// TwinCAT 3 PLC project TEXXX_XXX
// ProgramVersion: 3.1.4024.0
// libraries:
//   Tc2_Standard, * (Beckhoff Automation GmbH)
//   Tc2_System, * (Beckhoff Automation GmbH)
//   Tc2_Utilities, * (Beckhoff Automation GmbH)
//   Tc3_Module, * (Beckhoff Automation GmbH)
// project tree:
//   DUTs/HMI/ ST_StatusBanner.TcDUT (not stored)
//   DUTs/IO/CARDS/ ST_Terminal_Info.TcDUT, ST_EL1809.TcDUT, ST_EL2809.TcDUT
//   DUTs/MASTER/ E_MachineState.TcDUT, E_ProcessCycle.TcDUT, ST_ButtonsLamps.TcDUT (not stored), ST_HMI_IO.TcDUT, ST_MachineStatus.TcDUT, ST_MasterCTRL.TcDUT, ST_StationCMD.TcDUT, ST_StationStatus.TcDUT (not stored), ST_Puls.TcDUT (not stored), ST_StatisticsHMI.TcDUT (not stored)
//   DUTs/MASTER/log_CSV/ ST_CSVProcess.TcDUT, ST_UserLog.TcDUT (not stored), ST_CycleData.TcDUT
//   DUTs/STATIONS/STATION_1/ E_Station1_State.TcDUT, ST_CycleDataStation1.TcDUT, ST_Station_1.TcDUT
//   DUTs/STATIONS/STATION_2/ E_Station2_State.TcDUT, ST_CycleDataStation2.TcDUT, ST_Station_2.TcDUT
//   DUTs/STATIONS/STATION_3/ E_Station3_State.TcDUT, ST_CycleDataStation3.TcDUT, ST_Station_3.TcDUT
//   DUTs/USER_ALARMS_EVENTS/EVENTS/ ST_ActiveEvents.TcDUT (not stored), ST_EventsAssigment.TcDUT, ST_EventsAssigmentGeneral.TcDUT, ST_EventsHistory.TcDUT, ST_EVENT.TcDUT, ST_StationEvents.TcDUT
//   DUTs/USER_ALARMS_EVENTS/ ST_UserLogHMI.TcDUT (not stored)
//   GVLs/ GVL_Constants.TcGVL, GVL_HMI.TcGVL, GVL_IO.TcGVL, GVL_Master.TcGVL, GVL_Persistent.TcGVL, GVL_Stations.TcGVL
//   / PlcTask.TcTTO (not stored)
//   POUs/A_MASTER/ A_1_PRG_Main_Master.TcPOU, A_2_PRG_MachineCtrl.TcPOU, A_3_PRG_FaultHandling.TcPOU, A_4_PRG_MasterSystemTime.TcPOU
//   POUs/B_STATIONS/B_1_STATION_1/ B_1_1_PRG_Master_Station_1.TcPOU
//   POUs/B_STATIONS/B_2_STATION_2/ B_2_1_PRG_Master_Station_2.TcPOU
//   POUs/B_STATIONS/B_3_STATION_3/ B_3_1_PRG_Master_Station_3.TcPOU
//   POUs/C_HMI/ C_1_PRG_MainHMI.TcPOU
//   POUs/D_CSV/ D_1_WriteDataToCSV.TcPOU
//   POUs/ MAIN.TcPOU
//   POUs/Utilities/ FB_EventsManager.TcPOU, FB_UserLog.TcPOU, FB_Pulse.TcPOU (not stored), FB_TerminalInfo.TcPOU, FB_TimeControl.TcPOU, PRG_Puls.TcPOU (not stored)
// real-time tasks:
//   TASK PlcTask: cycle T#10ms, priority 20, ADS port 350

// ---- DUTs/IO/CARDS/ST_Terminal_Info.TcDUT
TYPE ST_Terminal_Info :
STRUCT
	
	nTerminal_State                        AT %I*			:    UINT;	// Terminal State from IO Terminal Info Data
	sTerminalInfo                                           :    STRING;
    fbTerminalInfo                                          :    FB_TerminalInfo;
END_STRUCT
END_TYPE

// ---- DUTs/IO/CARDS/ST_EL1809.TcDUT
TYPE ST_EL1809 :
STRUCT
	//--------------------------------------------------------------------------------------------------------
	sTerminalName                                           :   STRING(200):= 'EL1809 | 16-Channel Digital Input';
    //============================================================================================================================	
	// TERMINAL - EL1809 16-Channel Digital Input Terminal 	
	iEL1809_Ch1                				AT %I*			: 	BOOL;	// EL1809 channel 1
	iEL1809_Ch2                   			AT %I*			: 	BOOL;	// EL1809 channel 2
	iEL1809_Ch3        						AT %I*	 		: 	BOOL;	// EL1809 channel 3
	iEL1809_Ch4   							AT %I*	 		: 	BOOL;	// EL1809 channel 4
	iEL1809_Ch5         				 	AT %I*	 		: 	BOOL;	// EL1809 channel 5 		     			
	iEL1809_Ch6 							AT %I*			: 	BOOL;	// EL1809 channel 6
	iEL1809_Ch7               				AT %I*          :   BOOL;   // EL1809 channel 7 
    iEL1809_Ch8          					AT %I*          :   BOOL;   // EL1809 channel 8
    iEL1809_Ch9           					AT %I*          :   BOOL;   // EL1809 channel 9
	iEL1809_Ch10                			AT %I*          :   BOOL;   // EL1809 channel 10
	iEL1809_Ch11                    		AT %I*          :   BOOL;   // EL1809 channel 11
	iEL1809_Ch12                          	AT %I*          :   BOOL;   // EL1809 channel 12	   
	iEL1809_Ch13         		    		AT %I*	 		: 	BOOL;	// EL1809 channel 13   
	iEL1809_Ch14       						AT %I*	 		: 	BOOL;	// EL1809 channel 14 
	iEL1809_Ch15							AT %I*			: 	BOOL;	// EL1809 channel 15  
	iEL1809_Ch16							AT %I*	 		: 	BOOL;	// EL1809 channel 16  	
	
	stTerminalInfo											: 	ST_Terminal_Info;

END_STRUCT
END_TYPE

// ---- DUTs/IO/CARDS/ST_EL2809.TcDUT
TYPE ST_EL2809 :
STRUCT
	//--------------------------------------------------------------------------------------------------------
	sTerminalName                                           :   STRING(200):= 'EL2809 | 16-Channel Digital Output';
	//=============================================================================================================
	// TERMINAL - EL2809	16-Channel Digital Output Terminal	 (Term ...)
	qiEL2809_Ch1 							AT %Q*			: 	BOOL;	// EL2809 channel 1
	qiEL2809_Ch2							AT %Q* 			: 	BOOL;	// EL2809 channel 2
	qiEL2809_Ch3             				AT %Q*	 		: 	BOOL;	// EL2809 channel 3 			
	qiEL2809_Ch4      						AT %Q*	 		: 	BOOL;	// EL2809 channel 4 
	qiEL2809_Ch5  							AT %Q*	 		: 	BOOL;	// EL2809 channel 5
	qiEL2809_Ch6 							AT %Q*	 		: 	BOOL;	// EL2809 channel 6 	
	qiEL2809_Ch7         		    		AT %Q*			: 	BOOL;	// EL2809 channel 7	
	qiEL2809_Ch8							AT %Q*	 		: 	BOOL;	// EL2809 channel 8	
	qiEL2809_Ch9                 			AT %Q*          :   BOOL;   // EL2809 channel 9
	qiEL2809_Ch10             				AT %Q*          :   BOOL;   // EL2809 channel 10   	
	qiEL2809_Ch11     						AT %Q*	 		: 	BOOL;	// EL2809 channel 11	
	qiEL2809_Ch12   						AT %Q*	 		: 	BOOL;	// EL2809 channel 12 
    qiEL2809_Ch13 			        		AT %Q*	 		: 	BOOL;	// EL2809 channel 13 
	qiEL2809_Ch14                 			AT %Q*	 		: 	BOOL;	// EL2809 channel 14 
	qiEL2809_Ch15							AT %Q*	 		: 	BOOL;	// EL2809 channel 15 
    qiEL2809_Ch16         		        	AT %Q*	 		: 	BOOL;	// EL2809 channel 16  
	
	stTerminalInfo											: 	ST_Terminal_Info;
	
END_STRUCT
END_TYPE

// ---- DUTs/MASTER/E_MachineState.TcDUT
{attribute 'qualified_only'}
{attribute 'strict'}
TYPE E_MachineState :
(
	SYSTEM_POWER_UP			:=0,
	IMMEDIATE_STOPPED		:=100,
	SYSTEM_INITIALISING		:=110,
	SYSTEM_READY_TO_START	:=120,
	SYSTEM_AUTO_CYCLE		:=130,
	SYSTEM_STANDBY			:=140,
	STOPPING				:=150,
	CYCLE_STOPPED			:=160,
	MANUAL_MODE				:=170,
	IMMEDIATE_FAULT			:=190,
	CYCLE_STOP_FAULT		:=200
);
END_TYPE

// ---- DUTs/MASTER/E_ProcessCycle.TcDUT
{attribute 'qualified_only'}
{attribute 'strict'}
TYPE E_ProcessCycle :
(

	
IDLE								:=0,
STATION1_MOV1						:=10,
WAIT_STATION1_MOV1					:=20,
STATION2_MOV2						:=30,
WAIT_STATION2_MOV2					:=40,
STATION3_MOV3						:=50,
WAIT_STATION3_MOV3					:=60,
STATION1_MOV3_STATION2_MOV2			:=70,
WAIT_STATION1_MOV3_STATION2_MOV2	:=80,
SAVE_DATA							:=90,
SAVE_DATA2							:=100,
CSV									:=110,

RESET_ALL_CMD						:=120

);
END_TYPE

// ---- DUTs/MASTER/log_CSV/ST_CSVProcess.TcDUT
TYPE ST_CSVProcess :
STRUCT
	
	//INPUTS
	bWriteData			: BOOL;
	sFileNamePath		: STRING(255);
	sDate				: STRING(255);
	aDataHistoryArrayLength : DINT;
	nMAX_CSV_ROWS		: UDINT;
	nMAX_CSV_COLUMNS	: UDINT;
	nDataHistoryIndex	: DINT;
	

	//OUTPUTS
	bError				: BOOL;
	bBusy				: BOOL;
	bDataWrited			: BOOL;
	
	
	
	
END_STRUCT
END_TYPE

// ---- DUTs/MASTER/log_CSV/ST_CycleData.TcDUT
TYPE ST_CycleData :
STRUCT
//-----------------------------------------------------------------------------------GENERAL------------------------------------------------------------------------------------//	

	bPass				: BOOL;
	bFail				: BOOL;	
	sData				: STRING;	
	sTime				: STRING;
	
//-----------------------------------------------------------------------------------STATION 1------------------------------------------------------------------------------------//
/////////////////////////////////////////////////////////////////////////////////////SETTINGS/////////////////////////////////////////////////////////////////////////////////////			
(**************************************************************************CURRENT SETTINGS DURING CYCLE. VELOCITY FOR EXAMPLE****************************************************)	
	
	sSetting1_1			: STRING;	
	nSetting2_1			: DINT;
	bSetting3_1			: BOOL;
	
/////////////////////////////////////////////////////////////////////////////////////GENERAL DATA/////////////////////////////////////////////////////////////////////////////////////			
(**************************************************************************RESULT DATA OF THE CYCLE. DISTANCE FOR EXAMPLE************************************************************)	
	
	sDATA1_1			: STRING;
	nDATA2_1			: DINT;
	bDATA3_1			: BOOL;

////////////////////////////////////////////////////////////////////////////////////RESULTS////////////////////////////////////////////////////////////////////////////////////////
(**************************************************************************DETERMINE IF THE PART FAIL OR PASS*********************************************************************)

	bPass_1				: BOOL;
	bFail_1				: BOOL;		


	
	
	
//-----------------------------------------------------------------------------------STATION 2------------------------------------------------------------------------------------//
/////////////////////////////////////////////////////////////////////////////////////SETTINGS/////////////////////////////////////////////////////////////////////////////////////			
(**************************************************************************CURRENT SETTINGS DURING CYCLE. VELOCITY FOR EXAMPLE****************************************************)	
	
	sSetting1_2			: STRING;	
	nSetting2_2			: DINT;
	bSetting3_2			: BOOL;
	
/////////////////////////////////////////////////////////////////////////////////////GENERAL DATA/////////////////////////////////////////////////////////////////////////////////////			
(**************************************************************************RESULT DATA OF THE CYCLE. DISTANCE FOR EXAMPLE************************************************************)	
	
	sDATA1_2			: STRING;
	nDATA2_2			: DINT;
	bDATA3_2			: BOOL;

////////////////////////////////////////////////////////////////////////////////////RESULTS////////////////////////////////////////////////////////////////////////////////////////
(**************************************************************************DETERMINE IF THE PART FAIL OR PASS*********************************************************************)

	bPass_2				: BOOL;
	bFail_2				: BOOL;		
	
	
	
	
	
//-----------------------------------------------------------------------------------STATION 3------------------------------------------------------------------------------------//
/////////////////////////////////////////////////////////////////////////////////////SETTINGS/////////////////////////////////////////////////////////////////////////////////////			
(**************************************************************************CURRENT SETTINGS DURING CYCLE. VELOCITY FOR EXAMPLE****************************************************)	
	
	sSetting1_3			: STRING;	
	nSetting2_3			: DINT;
	bSetting3_3			: BOOL;
	
/////////////////////////////////////////////////////////////////////////////////////GENERAL DATA/////////////////////////////////////////////////////////////////////////////////////			
(**************************************************************************RESULT DATA OF THE CYCLE. DISTANCE FOR EXAMPLE************************************************************)	
	
	sDATA1_3			: STRING;
	nDATA2_3			: DINT;
	bDATA3_3			: BOOL;

////////////////////////////////////////////////////////////////////////////////////RESULTS////////////////////////////////////////////////////////////////////////////////////////
(**************************************************************************DETERMINE IF THE PART FAIL OR PASS*********************************************************************)

	bPass_3				: BOOL;
	bFail_3				: BOOL;		
	



	
	
END_STRUCT
END_TYPE

// ---- DUTs/MASTER/ST_HMI_IO.TcDUT
TYPE ST_HMI_IO :
STRUCT
	
	bTriggerButtonA				:BOOL;
	bTriggerButtonB				:BOOL;
	bTriggerButtonC				:BOOL;
	
	bOutPutSigA					:BOOL;
	bOutPutSigB					:BOOL;
	bOutPutSigC					:BOOL;
	
END_STRUCT
END_TYPE

// ---- DUTs/MASTER/ST_MachineStatus.TcDUT
TYPE ST_MachineStatus :
STRUCT
	////////////////////////////:
	eMachineState				:E_MachineState;
	
	// Status Flags:
	bSystemPowerUp 				:BOOL;
	bImmediateStopped 			:BOOL;
	bInitialising 				:BOOL;
	bReadyToStart 				:BOOL;
	bAutoCycle 					:BOOL;
	bStandby					:BOOL;
	bStopping					:BOOL;	
	bCycleStopped 				:BOOL;
	bImmediateFault 			:BOOL;
	bCycleStopFault 			:BOOL;
	bManualMode					:BOOL;

END_STRUCT
END_TYPE

// ---- DUTs/MASTER/ST_MasterCTRL.TcDUT
TYPE ST_MasterCTRL :
STRUCT
	

	// Request Flags
	bManualModeRequest					:BOOL;
	
	bCycleStopRequest					:BOOL;
	
	bNoImmediateFault					:BOOL;
	bNoCycleStopFault					:BOOL;


	// Feedback Flags
	bAllStationsReady					:BOOL;
	bAllStationsStopped					:BOOL;
	
	bPowerUpTimerComplete				:BOOL;

	
//-------------------------------------------------------------------------------oldschoo1
		
END_STRUCT
END_TYPE

// ---- DUTs/MASTER/ST_StationCMD.TcDUT
TYPE ST_StationCMD :
STRUCT
//Universal Module CMD Struct

    bEnable       			:BOOL;	// Request module to activate devices
	bExecute				:BOOL;	// Request module to execute CMD
    bReset        			:BOOL;	// Request module to reset error or state
    bAbort        			:BOOL;	// Emergency stop or cancel current task
	bReady					:BOOL;	// Get ready
	bEndCycle				:BOOL; // End cycle
	
	nTaskID       			:UINT;	// Request a Task by its ID	
    bManualMode   			:BOOL;	// Request Manual Mode(jog mode)
	
	
END_STRUCT
END_TYPE

// ---- DUTs/STATIONS/STATION_1/E_Station1_State.TcDUT
{attribute 'qualified_only'}
{attribute 'strict'}
TYPE E_Station1_State :
(
	//GENERIC
	ABORTED				:=10,
	RESET_ERROR			:=20,
	HOMING				:=30,
	READY				:=40,
	//MANUAL_MODE		:=50, /manual mode not needed.
	ERROR				:=60,
	PERSISTENT_ERROR	:=70,
	STOPPING			:=80,
	//SPECIFIC FOR EVERY STATION
	MOVEMENT_A			:=100,
	MOVEMENT_B			:=120,
	MOVEMENT_C			:=130,
	DONE				:=140,
	RESULTS				:=160,
	RESET				:=180
);
END_TYPE

// ---- DUTs/STATIONS/STATION_1/ST_CycleDataStation1.TcDUT
TYPE ST_CycleDataStation1 :
STRUCT
	/////////////////////////////////////////////////////////////////////////////////////SETTINGS/////////////////////////////////////////////////////////////////////////////////////			
(**************************************************************************CURRENT SETTINGS DURING CYCLE. VELOCITY FOR EXAMPLE****************************************************)	
	
	sSetting1			: STRING;	
	nSetting2			: DINT;
	bSetting3			: BOOL;
	
/////////////////////////////////////////////////////////////////////////////////////GENERAL DATA/////////////////////////////////////////////////////////////////////////////////////			
(**************************************************************************RESULT DATA OF THE CYCLE. DISTANCE FOR EXAMPLE************************************************************)	
	
	sDATA1				: STRING;
	nDATA2				: DINT;
	bDATA3				: BOOL;

////////////////////////////////////////////////////////////////////////////////////RESULTS////////////////////////////////////////////////////////////////////////////////////////
(**************************************************************************DETERMINE IF THE PART FAIL OR PASS*********************************************************************)

	bPass				: BOOL;
	bFail				: BOOL;		

END_STRUCT
END_TYPE

// ---- DUTs/STATIONS/STATION_1/ST_Station_1.TcDUT
TYPE ST_Station_1 :
STRUCT
	
	Mov1				: BOOL;		
	Mov2				: BOOL;	
	Mov3				: BOOL;		
	
END_STRUCT
END_TYPE

// ---- DUTs/STATIONS/STATION_2/E_Station2_State.TcDUT
{attribute 'qualified_only'}
{attribute 'strict'}
TYPE E_Station2_State :
(
		//GENERIC
	ABORTED				:=10,
	RESET_ERROR			:=20,
	HOMING				:=30,
	READY				:=40,
	//MANUAL_MODE			:=50, /manual mode not needed.
	ERROR				:=60,
	PERSISTENT_ERROR	:=70,
	STOPPING			:=80,
	//SPECIFIC FOR EVERY STATION
	MOVEMENT_A			:=100,
	MOVEMENT_B			:=120,
	MOVEMENT_C			:=130,
	DONE				:=140,
	RESULTS				:=160,
	RESET				:=180
);
END_TYPE

// ---- DUTs/STATIONS/STATION_2/ST_CycleDataStation2.TcDUT
TYPE ST_CycleDataStation2 :
STRUCT
	/////////////////////////////////////////////////////////////////////////////////////SETTINGS/////////////////////////////////////////////////////////////////////////////////////			
(**************************************************************************CURRENT SETTINGS DURING CYCLE. VELOCITY FOR EXAMPLE****************************************************)	
	
	sSetting1			: STRING;	
	nSetting2			: DINT;
	bSetting3			: BOOL;
	
/////////////////////////////////////////////////////////////////////////////////////GENERAL DATA/////////////////////////////////////////////////////////////////////////////////////			
(**************************************************************************RESULT DATA OF THE CYCLE. DISTANCE FOR EXAMPLE************************************************************)	
	
	sDATA1				: STRING;
	nDATA2				: DINT;
	bDATA3				: BOOL;

////////////////////////////////////////////////////////////////////////////////////RESULTS////////////////////////////////////////////////////////////////////////////////////////
(**************************************************************************DETERMINE IF THE PART FAIL OR PASS*********************************************************************)

	bPass				: BOOL;
	bFail				: BOOL;		

END_STRUCT
END_TYPE

// ---- DUTs/STATIONS/STATION_2/ST_Station_2.TcDUT
TYPE ST_Station_2 :
STRUCT
	
	Mov1				: BOOL;		
	Mov2				: BOOL;	
	Mov3				: BOOL;		
	
END_STRUCT
END_TYPE

// ---- DUTs/STATIONS/STATION_3/E_Station3_State.TcDUT
{attribute 'qualified_only'}
{attribute 'strict'}
TYPE E_Station3_State :
(
		//GENERIC
	ABORTED				:=10,
	RESET_ERROR			:=20,
	HOMING				:=30,
	READY				:=40,
	//MANUAL_MODE			:=50, /manual mode not needed.
	ERROR				:=60,
	PERSISTENT_ERROR	:=70,
	STOPPING			:=80,
	//SPECIFIC FOR EVERY STATION
	MOVEMENT_A			:=100,
	MOVEMENT_B			:=120,
	MOVEMENT_C			:=130,
	DONE				:=140,
	RESULTS				:=160,
	RESET				:=180
);
END_TYPE

// ---- DUTs/STATIONS/STATION_3/ST_CycleDataStation3.TcDUT
TYPE ST_CycleDataStation3 :
STRUCT
	/////////////////////////////////////////////////////////////////////////////////////SETTINGS/////////////////////////////////////////////////////////////////////////////////////			
(**************************************************************************CURRENT SETTINGS DURING CYCLE. VELOCITY FOR EXAMPLE****************************************************)	
	
	sSetting1			: STRING;	
	nSetting2			: DINT;
	bSetting3			: BOOL;
	
/////////////////////////////////////////////////////////////////////////////////////GENERAL DATA/////////////////////////////////////////////////////////////////////////////////////			
(**************************************************************************RESULT DATA OF THE CYCLE. DISTANCE FOR EXAMPLE************************************************************)	
	
	sDATA1				: STRING;
	nDATA2				: DINT;
	bDATA3				: BOOL;

////////////////////////////////////////////////////////////////////////////////////RESULTS////////////////////////////////////////////////////////////////////////////////////////
(**************************************************************************DETERMINE IF THE PART FAIL OR PASS*********************************************************************)

	bPass				: BOOL;
	bFail				: BOOL;		

END_STRUCT
END_TYPE

// ---- DUTs/STATIONS/STATION_3/ST_Station_3.TcDUT
TYPE ST_Station_3 :
STRUCT
	
	Mov1				: BOOL;		
	Mov2				: BOOL;	
	Mov3				: BOOL;		
	
END_STRUCT
END_TYPE

// ---- DUTs/USER_ALARMS_EVENTS/EVENTS/ST_EventsAssigment.TcDUT
TYPE ST_EventsAssigment :
STRUCT
	
	sEventText							: STRING(255);
	sSolution							: STRING(255);
END_STRUCT
END_TYPE

// ---- DUTs/USER_ALARMS_EVENTS/EVENTS/ST_EventsAssigmentGeneral.TcDUT
TYPE ST_EventsAssigmentGeneral :
STRUCT
	
	astImmediateFaultEvents				: ARRAY [1..100] OF ST_EventsAssigment;
	astCycleStopFaultEvents				: ARRAY [1..100] OF ST_EventsAssigment;
	astCycleStopRequestEvents			: ARRAY [1..100] OF ST_EventsAssigment;
	astMessage							: ARRAY [1..100] OF ST_EventsAssigment;
	
	
END_STRUCT
END_TYPE

// ---- DUTs/USER_ALARMS_EVENTS/EVENTS/ST_EventsHistory.TcDUT
TYPE ST_EventsHistory :
STRUCT
	
	sEventTex									: STRING(255);
	sType										: STRING(255);
	sDate										: STRING(255);
	sTime										: STRING(255);
	abType										: DINT;					//1:Alarm
																		//2:Alert
																		//3:Message
	
END_STRUCT
END_TYPE

// ---- DUTs/USER_ALARMS_EVENTS/EVENTS/ST_EVENT.TcDUT
TYPE ST_EVENT :
STRUCT
	
	bImmediateFault						: BOOL;
	bCycleStopFault						: BOOL;
	bCycleStopRequest					: BOOL;
	bMessage							: BOOL;
	
	bAssignedID							: DINT;
	
	bEventFlag							: BOOL;
	bEventTimer							: TON;
	bEventText							: STRING(255);
	bEventTextHMI						: STRING(255);
	sSolution							: STRING(255);
	bActive								: BOOL;

END_STRUCT
END_TYPE

// ---- DUTs/USER_ALARMS_EVENTS/EVENTS/ST_StationEvents.TcDUT
TYPE ST_StationEvents :
STRUCT
	
	aEvents								: ARRAY [0..100] OF ST_EVENT;	
	
	bImmediateFault						: BOOL;
	bCycleStopFault						: BOOL;
	bCycleStopRequest					: BOOL;
			
END_STRUCT
END_TYPE

// ---- GVLs/GVL_Constants.TcGVL
VAR_GLOBAL CONSTANT
////////////////////////////////////////:	///////////////////////////////////////////////////
/////////////////////////////////////////////////////////////////////////////////////HMI/////////////////////////////////////////////////////////////////////////////////////
	
    sWHITE                              :   STRING(40)  := '{"color":"rgba(255,255,255,255)"}';
    sBLACK                              :   STRING(40)  := '{"color":"rgba(0,0,0,1)"}';
    sYELLOW                             :   STRING(40)  := '{"color":"rgba(255,255,0,1)"}';
    sGREEN                             	:   STRING(40)  := '{"color":"rgba(70,166,63,1)"}';
	sLGREEN                             :   STRING(40)  := '{"color":"rgba(58,211,20,1)"}';
    sORANGE                             :   STRING(40)  := '{"color":"rgba(255,153,51,1)"}';
    sNYPROORANGE                        :   STRING(40)  := '{"color":"rgba(255,140,0,1)"}';
    sRED                                :   STRING(40)  := '{"color":"rgba(255,0,0,1)"}';
	sLRED                               :   STRING(40)  := '{"color":"rgba(233,53,44,1)"}';
    sBLUE                               :   STRING(40)  := '{"color":"rgba(0,0,255,1)"}';
	sLBLUE                              :   STRING(40)  := '{"color":"rgba(0,162,232,1)"}';
    sGREY                               :   STRING(40)  := '{"color":"rgba(164,158,158,1)"}';
    sScreenGREY                         :   STRING(40)  := '{"color":"rgba(225,225,225,1)"}';
    sDARKGREY                           :   STRING(40)  := '{"color":"rgba(50,50,50,1)"}';
    sPURPLE                             :   STRING(40)  := '{"color":"rgba(128,0,128,1)"}';
    sVIOLET                             :   STRING(40)  := '{"color":"rgba(204,153,255,1)"}';
    sTRANSP                             :   STRING(40)  := '{"color":"rgba(255,255,255,0)"}';
    sGREENPass                          :   STRING(40)  := '{"color":"rgba(0,153,51,1)"}';
    sREDFail                            :   STRING(40)  := '{"color":"rgba(244,68,68,255)"}';
    sBLUEInProgress                     :   STRING(40)  := '{"color":"rgba(54,100,221,1)"}';
	sGREENISHTEAColor					:	STRING(40)  := '{"color":"rgba(60,192,134,255)"}'	;		

	nBLACK								: 	DWORD 	:= 	16#FF000000;	 // format: TTRRGGBB where T -> 00 = full transparency and FF = full opaque
	nWHITE								: 	DWORD 	:= 	16#FFFFFFFF;
	nYELLOW								: 	DWORD 	:= 	16#FFFFFF00; 
	nGREEN								: 	DWORD 	:= 	16#FF008A00;
	nLIGHTGREEN                         :   DWORD   :=  16#FF98FB89;
	nORANGE								: 	DWORD 	:= 	16#FFFFA500;
	nNYPROORANGE						:	DWORD	:=	16#FFF05322;
	nRED								: 	DWORD 	:= 	16#FFFF0000;
	nBLUE								: 	DWORD 	:= 	16#FF0000FF;
	nLIGHTBLUE                          :   DWORD   :=  16#FF08ADF4;
	nGREY								: 	DWORD 	:= 	16#FFA9A9A9;	
	nDARKGREY							:	DWORD	:=	16#FF808080;
	nPURPLE								:	DWORD	:=	16#FF800080;
	nVIOLET								:	DWORD	:=	16#FFEE82EE;
	nTRANSP								:	DWORD	:=	16#00FFFFFF;	// full transparent WHITE
	
/////////////////////////////////////////////////////////////////////////////////////CSV/////////////////////////////////////////////////////////////////////////////////////
	
	MAX_CSV_ROWS 						: UDINT := 200;
	MAX_CSV_COLUMNS 					: UDINT := 27;
	MAX_CSV_FIELD_LENGTH				: UDINT := 100;
	
	
	
END_VAR

// ---- GVLs/GVL_HMI.TcGVL
VAR_GLOBAL
////////////////////////////////////////:	///////////////////////////////////////////////////
/////////////////////////////////////////////////////////////////////////////////////GENERIC/////////////////////////////////////////////////////////////////////////////////////

	stHMI_IO							: ST_HMI_IO;
	bQuitHMI							: BOOL;
	bShutDown							: BOOL;
	stStatusBanner						: ST_StatusBanner;
	

/////////////////////////////////////////////////////////////////////////////////////SYSTEM INFO/////////////////////////////////////////////////////////////////////////////////////

	sSoftwareVersion					: STRING := ' 1.0 ';
	sSoftwareDate						: STRING := ' 10.December.2024 ';
	sTC3Version							: STRING := ' v3.1.4024.53, Runtime v3.1.4024.40 ';
	sHMIVersion							: STRING := ' TcXaeShell Version 15.0.28010.2050 D15.8 ';
	sSystemName							: STRING := ' Print & Applay Labeller ' ;
	sProjectID							: STRING := ' TE 1099 PAL' ;
	sAplication                     	: STRING := ' Print & Applay Labeller ';
	sHMIServer                			: STRING := ' ---- ';
	
	NetAmsId        	       			: T_AmsNetId := ''; // AMS-ID for com port setup 
	
/////////////////////////////////////////////////////////////////////////////////////USER LOG/////////////////////////////////////////////////////////////////////////////////////

	sUserGroupIn						: STRING;
	sUserGroupOut						: STRING;
	sUserName							: STRING;
	bUserLoggedIn						: BOOL;			
	bLogOut								: BOOL;	
	rUserLoggedIn						: R_TRIG;

/////////////////////////////////////////////////////////////////////////////////////MANUAL/////////////////////////////////////////////////////////////////////////////////////

	bEnableManual						: BOOL;
	nMainRegion							: DINT;
	bManualModeOffFlag					: BOOL;
	
END_VAR

// ---- GVLs/GVL_IO.TcGVL
VAR_GLOBAL
	
	

	//	dw_T01_EK1100                                                	| EtherCAT Coupler 
	//	dw_T02_EL6070-0033                                           	| EtherCAT Terminal, license key for TwinCAT 3.1
	
	dw_T03_EL1809                                                		: st_EL1809; //16 Channel Digital Input ( 24VDC ) 
	dw_T04_EL2809                                                		: st_EL2809; // 16 Channel Digital Output ( 24VDC )

END_VAR

// ---- GVLs/GVL_Master.TcGVL
VAR_GLOBAL
////////////////////////////////////////:	///////////////////////////////////////////////////
/////////////////////////////////////////////////////////////////////////////////////GENERIC/////////////////////////////////////////////////////////////////////////////////////

	// PowerUP 
	tonSystemPowerUP				:TON;
	tSystemPowerUP_Time				:TIME								:=T#35S;
	bSystemPoweringUP				:BOOL								:=TRUE; //Global System PowerUP Flag
	
	fbSystemShutDown     	        : NT_Shutdown;
	stButtonsLamps					: ST_ButtonsLamps;
	stPuls							: ST_Puls;		

	stCSVProcess					: ST_CSVProcess;
/////////////////////////////////////////////////////////////////////////////////////Event Log/////////////////////////////////////////////////////////////////////////////////////
	
	stStationEvents				: ARRAY[0..3] OF  ST_StationEvents;//0: GENERAL
																	//1: STATION 1
																	//1: STATION 2
																	//3: STATION 3
	astActiveEvents				: ARRAY [0..50] OF ST_ActiveEvents;
	astEventsHistory			: ARRAY[0..200] OF ST_EventsHistory;
	
/////////////////////////////////////////////////////////////////////////////////////MACHINE CONTROL////////////////////////////////////////////////////////////////////////////
	
	stMachineStatus					: ST_MachineStatus;	
	stMasterCtrl					: ST_MasterCTRL;
	bStatisticsTest					: ARRAY[0..6] OF  BOOL;
	
////////////////////////////////////////////////////////////////////////////////////SYSTEM////////////////////////////////////////////////////////////////////////////
	stSystemTime				: TIMESTRUCT;
	sSystemTime					: STRING(255);
	sSystemDate					: STRING(255);
	
	bResetTest								: BOOL;
	tonResetTest							: TON;
	
	stEventsAssigment						: ST_EventsAssigmentGeneral;	
END_VAR

// ---- GVLs/GVL_Persistent.TcGVL

VAR_GLOBAL PERSISTENT
	
/////////////////////////////////////////////////////////////////////////////////////Log/////////////////////////////////////////////////////////////////////////////////////
	
	stUserLog					: ARRAY [0..250] OF ST_UserLog;
	
	stStatisticsHMI				: ARRAY [0..3] OF ST_StatisticsHMI;	//0: GENERAL
																	//1: STATION 1
																	//2: STATION 2
																	//3: STATION 3
	aDataHistory				: ARRAY[0..200] OF ST_CycleData;
	nIndexDataHistory			: DINT;


END_VAR

// ---- GVLs/GVL_Stations.TcGVL
VAR_GLOBAL
/////////////////////////////////////////////////////////////////////////////////////Station 1/////////////////////////////////////////////////////////////////////////////////////
	
	stStation1							: ST_Station_1;
	CMD_Station1						: ST_StationCMD;
	stCycleDataStation1					: ST_CycleDataStation1;
	
/////////////////////////////////////////////////////////////////////////////////////Station 2/////////////////////////////////////////////////////////////////////////////////////

	stStation2							: ST_Station_2;
	CMD_Station2						: ST_StationCMD;
	stCycleDataStation2					: ST_CycleDataStation2;

/////////////////////////////////////////////////////////////////////////////////////Station 3/////////////////////////////////////////////////////////////////////////////////////

	stStation3							: ST_Station_3;	
	CMD_Station3						: ST_StationCMD;
	stCycleDataStation3					: ST_CycleDataStation3;

END_VAR

// ---- POUs/A_MASTER/A_1_PRG_Main_Master.TcPOU
PROGRAM A_1_PRG_Main_Master
VAR
	
	rtrigButton             				: ARRAY[1..3] OF Tc2_Standard.R_TRIG;
	ftrigButton             				: ARRAY[1..3] OF Tc2_Standard.F_TRIG; 
	
	fbStringFormatter       				: Tc2_Utilities.FB_FormatString;
	fbEventsManager							: FB_EventsManager;
	
	ntShutdown								: TC2_Utilities.NT_Shutdown;
	closeChrome 							: NT_StartProcess;
	tonUserLogOut							: TON;
	fbUserLog								: FB_UserLog;
	
	nFindAdm								: INT;
	nFindEng								: INT;
	nFindOpe								: INT;
	sUserGroupName							: STRING (255);
	sAdmGroup								: STRING (255)							:= 'Administrator';
	sEngGroup								: STRING (255)							:= 'Engineer';
	sOpeGroup								: STRING (255)							:= 'Operator';
	
	rEfficency								: STRING(510);
	
	fbSystemTime							: NT_GetTime;
	

	
END_VAR

/////////////////////////////////////////////////////////////////////////////////////GENERAL/////////////////////////////////////////////////////////////////////////////////////
A_3_PRG_FaultHandling();
a_ACT_ButtonsLamps();
d_ACT_ShutdownAndQuit();
e_ACT_UserLog();
f_ACT_TerminalInfo();
g_ACT_Manual();
h_ACT_Statistics();

C_1_PRG_MainHMI();
D_1_WriteDataToCSV();

PRG_Puls();

// System PowerUP CTRL
tonSystemPowerUP(IN:=bSystemPoweringUP, PT:=tSystemPowerUP_Time);
IF tonSystemPowerUP.Q THEN 
bSystemPoweringUP:=FALSE;
END_IF


A_4_PRG_MasterSystemTime();
/////////////////////////////////////////////////////////////////////////////////////STATIONS/////////////////////////////////////////////////////////////////////////////////////

B_1_1_PRG_Master_Station_1(CMD := CMD_Station1);
B_2_1_PRG_Master_Station_2(CMD := CMD_Station2);
B_3_1_PRG_Master_Station_3(CMD := CMD_Station3);

/////////////////////////////////////////////////////////////////////////////////////PROCESS/////////////////////////////////////////////////////////////////////////////////////

A_2_PRG_MachineCtrl();

/////////////////////////////////////////////////////////////////////////////////////EVENT LOG/////////////////////////////////////////////////////////////////////////////////////

fbEventsManager	(			//INPUTS
							bPulse 							:= stPuls.bFlash10Hz, 
							bResetFaults 					:= bResetTest, 
							stStationEvents 				:= stStationEvents,
							sSystemTime						:= sSystemTime,
							sSystemDate						:= sSystemDate,
 							stEventsAssigment				:= stEventsAssigment,
							
							//OUTPUTS
							astActiveEvents 				=> astActiveEvents,
							astEventsHistory				=> astEventsHistory
							);



////////////////////////////////////////////////////////////////////////////////////SYSTEM DATE & TIME/////////////////////////////////////////////////////////////////////////////////////

fbSystemTime( START := stPuls.bFlash10Hz, TIMESTR => stSystemTime);
	

sSystemTime					:= 	CONCAT( STR1 := WORD_TO_STRING(stSystemTime.wHour), STR2 := CONCAT( STR1 := ':', STR2 := 
								CONCAT( STR1 := WORD_TO_STRING(stSystemTime.wMinute), STR2 := 
								CONCAT(STR1 := ':', STR2 := WORD_TO_STRING(stSystemTime.wSecond)))));
								
sSystemDate					:= 	CONCAT( STR1 := WORD_TO_STRING(stSystemTime.wDay), STR2 := 
								CONCAT(STR1 := '/', STR2 := CONCAT(STR1 := WORD_TO_STRING(stSystemTime.wMonth), STR2 := 
								CONCAT(STR1 := '/', STR2 := WORD_TO_STRING(stSystemTime.wYear)))));

ACTION a_ACT_ButtonsLamps:
//===================================================================
stButtonsLamps.bStartButtonFallingEdge 	:= ftrigButton[1].Q ;
stButtonsLamps.bStartButtonRisingEdge 	:= rtrigButton[1].Q ;
stButtonsLamps.bStopButtonFallingEdge 	:= ftrigButton[2].Q ; 
stButtonsLamps.bStopButtonRisingEdge 	:= rtrigButton[2].Q ;  
stButtonsLamps.bResetButtonFallingEdge 	:= ftrigButton[3].Q ;
stButtonsLamps.bResetButtonRisingEdge 	:= rtrigButton[3].Q ;



ftrigButton[1](CLK :=);
rtrigButton[1](CLK						:=);
ftrigButton[2](CLK						:=);
rtrigButton[2](CLK						:=);
ftrigButton[3](CLK	:=bResetTest 		);
rtrigButton[3](CLK						:=);



//GVL_IO.dw_T11_EL2809.qRESETButton_Indicator := stPuls.bFlash2Hz AND (NOT stMachineStatus.bInitialising AND NOT stMachineStatus.bAutoCycle AND NOT stMachineStatus.bManualMode AND NOT stMachineStatus.bReadyToStart) ;
//GVL_IO.dw_T11_EL2809.qStartButton_Indicator := (stPuls.bFlash2Hz AND stMachineStatus.bReadyToStart) OR (stMachineStatus.bManualMode AND stPuls.bFlash4Hz ) ;
END_ACTION

ACTION d_ACT_ShutdownAndQuit:
closeChrome(
    NetId := '',
    PathStr := 'C:\Windows\System32\mshta vbscript:Execute("CreateObject(""WScript.Shell"").Run ""powershell -c',
    DirName := 'C:\Windows\System32\WindowsPowerShell\v1.0',
    ComndLine := 'taskkill /F /IM chrome.exe /T"", 0: window.close")',
    Start := bQuitHmi,
    TmOut := DEFAULT_ADS_TIMEOUT
);
 
bQuitHmi:= FALSE;

ntShutdown(NETID := NetAmsId, DELAY := 5, START := bShutDown);
END_ACTION

ACTION e_ACT_UserLog:
sUserGroupName																:= sUserGroupIn;

nFindAdm	:= TC2_Utilities.FIND( 	STR1									:= sUserGroupName,
									STR2									:= sAdmGroup);
									
nFindEng	:= TC2_Utilities.FIND( 	STR1									:= sUserGroupName,
									STR2									:= sEngGroup);
					
nFindOpe	:= TC2_Utilities.FIND( 	STR1									:= sUserGroupName,
									STR2									:= sOpeGroup);
				
IF nFindAdm <> 0 THEN
	sUserGroupOut															:= 'Administrator';
ELSIF nFindEng <> 0 THEN
	sUserGroupOut															:= 'Engineer';
ELSIF nFindOpe <> 0 THEN
	sUserGroupOut															:= 'Operator';
ELSE sUserGroupOut															:= '';
END_IF

tonUserLogOut( IN := (sUserGroupOut <> 'Administrator' OR sUserGroupOut <> 'Engineer') AND bUserLoggedIn , PT := T#10M);

IF tonUserLogOut.Q THEN
	bLogOut 											:= TRUE;
ELSE bLogOut 											:= FALSE;
END_IF

rUserLoggedIn( CLK := bUserLoggedIn);

fbUserLog(	nNumberOfData								:= 250,
			bSaveSignal									:= rUserLoggedIn.Q, 
			sUser										:= sUserName,
			sGroup										:= sUserGroupOut,
			sDate										:= sSystemDate,
			sTime										:= sSystemTime,
			aDataOutput									:= stUserLog);
END_ACTION

ACTION f_ACT_TerminalInfo:
dw_T03_EL1809.stTerminalInfo.fbTerminalInfo( 	nTerminalState						:= dw_T03_EL1809.stTerminalInfo.nTerminal_State,
												sTerminalState						=> dw_T03_EL1809.stTerminalInfo.sTerminalInfo);
												
dw_T04_EL2809.stTerminalInfo.fbTerminalInfo(	nTerminalState						:= dw_T04_EL2809.stTerminalInfo.nTerminal_State,
												sTerminalState						=> dw_T04_EL2809.stTerminalInfo.sTerminalInfo);
END_ACTION

ACTION g_ACT_Manual:


IF stMachineStatus.bReadyToStart THEN
	bEnableManual											:= TRUE;
ELSE bEnableManual											:= FALSE;
END_IF

IF nMainRegion = 5 AND stMasterCtrl.bNoImmediateFault AND stMasterCtrl.bNoCycleStopFault
	AND NOT stMasterCtrl.bCycleStopRequest AND NOT stButtonsLamps.bStopButtonFallingEdge THEN
	stMasterCtrl.bManualModeRequest							:= TRUE;
	bManualModeOffFlag										:= FALSE;
ELSE 
	stMasterCtrl.bManualModeRequest							:= FALSE; 
	bManualModeOffFlag										:= TRUE;											
END_IF
END_ACTION

ACTION h_ACT_Statistics:
stStatisticsHMI[0].sName			:= 'TOTAL';

stStatisticsHMI[0].nGood		:= stStatisticsHMI[1].nGood + stStatisticsHMI[2].nGood + stStatisticsHMI[3].nGood;
stStatisticsHMI[0].nTotalGood	:= stStatisticsHMI[1].nTotalGood + stStatisticsHMI[2].nTotalGood + stStatisticsHMI[3].nTotalGood;
stStatisticsHMI[0].nBad			:= stStatisticsHMI[1].nBad + stStatisticsHMI[2].nBad + stStatisticsHMI[3].nBad;
stStatisticsHMI[0].nTotalBad	:= stStatisticsHMI[1].nTotalBad + stStatisticsHMI[2].nTotalBad + stStatisticsHMI[3].nTotalBad;

								

IF (( stStatisticsHMI[0].nGood + stStatisticsHMI[0].nBad) <> 0) THEN
	
	rEfficency							:= LREAL_TO_FMTSTR(in := (DINT_TO_REAL(stStatisticsHMI[0].nGood) /( DINT_TO_REAL(stStatisticsHMI[0].nGood) + DINT_TO_REAL(stStatisticsHMI[0].nBad))) * 100.0,iPrecision := 2, bRound := TRUE);
	stStatisticsHMI[0].nEfficency		:= CONCAT(STR1 := '%', STR2 := (rEfficency));

ELSE stStatisticsHMI[0].nEfficency		:= CONCAT(STR1 := '%', STR2 := (DINT_TO_STRING(0)));
	
END_IF
END_ACTION

END_PROGRAM

// ---- POUs/Utilities/FB_EventsManager.TcPOU
FUNCTION_BLOCK FB_EventsManager

VAR_INPUT
	
	bPulse					: BOOL;
	sSystemTime				: STRING(255);
	sSystemDate				: STRING(255);

	
END_VAR

VAR_OUTPUT

	astActiveEvents			: ARRAY [0..50] OF ST_ActiveEvents;
	astEventsHistory		: ARRAY[0..200] OF ST_EventsHistory;;

END_VAR

VAR
	
	i								: ARRAY [0..1] OF DINT;
	j								: ARRAY [0..1] OF DINT;
	m								: ARRAY [0..3] OF DINT;
	k								: ARRAY [0..1] OF DINT;
	l								: DINT;
	n								: DINT;
	
	bEventsAssigmentSignal			: BOOL		:= TRUE;
	

	
END_VAR

VAR_IN_OUT
	
	stStationEvents			: ARRAY[0..3] OF ST_StationEvents;
	stEventsAssigment		: ST_EventsAssigmentGeneral;
	bResetFaults			: BOOL;
	
END_VAR

ACT_FaultTrig();
ACT_ActiveEvents_DataHistory();


IF bEventsAssigmentSignal THEN
	ACT_EventTextAssigment();
	bEventsAssigmentSignal := FALSE;
END_IF

ACTION ACT_ActiveEvents_DataHistory:
IF bPulse THEN

FOR k[0] := 0 TO 3 DO
	
	FOR k[1] := 0 TO 100 DO
		
		IF stStationEvents[k[0]].aEvents[k[1]].bImmediateFault AND stStationEvents[k[0]].aEvents[k[1]].bEventFlag AND NOT stStationEvents[k[0]].aEvents[k[1]].bActive THEN
			
			//ACTIVE EVENTS
			astActiveEvents[l].sEventTex				:= 	stStationEvents[k[0]].aEvents[k[1]].bEventTextHMI;
			astActiveEvents[l].sType					:= 'Immediate Fault';						
			astActiveEvents[l].abType					:= 1; 
			astActiveEvents[l].sSolution				:= stStationEvents[k[0]].aEvents[k[1]].sSolution;
			stStationEvents[k[0]].aEvents[k[1]].bActive := TRUE;
			
			//EVENTS HISTORY
			FOR n := 199 TO 0 BY -1 DO
							
				astEventsHistory[n+1].sEventTex				:= astEventsHistory[n].sEventTex;
				astEventsHistory[n+1].sType					:= astEventsHistory[n].sType;
				astEventsHistory[n+1].abType				:= astEventsHistory[n].abType;
				astEventsHistory[n+1].sDate					:= astEventsHistory[n].sDate;										
				astEventsHistory[n+1].sTime					:= astEventsHistory[n].sTime;
				
			END_FOR

			astEventsHistory[0].sEventTex				:= stStationEvents[k[0]].aEvents[k[1]].bEventTextHMI;
			astEventsHistory[0].sType					:= 'Immediate Fault';
			astEventsHistory[0].abType					:= 1;
			astEventsHistory[0].sDate					:= 	sSystemTime;										
			astEventsHistory[0].sTime					:= 	sSystemDate;
				
			l											:= l + 1;					
		END_IF
		
		IF stStationEvents[k[0]].aEvents[k[1]].bCycleStopFault AND stStationEvents[k[0]].aEvents[k[1]].bEventFlag AND NOT stStationEvents[k[0]].aEvents[k[1]].bActive THEN
			
			//ACTIVE EVENTS
			astActiveEvents[l].sEventTex				:= 	stStationEvents[k[0]].aEvents[k[1]].bEventTextHMI;
			astActiveEvents[l].sType					:= 'Cycle Stop Fault';						
			astActiveEvents[l].abType					:= 1; 
			astActiveEvents[l].sSolution				:= stStationEvents[k[0]].aEvents[k[1]].sSolution;
			stStationEvents[k[0]].aEvents[k[1]].bActive := TRUE;
			
			//EVENTS HISTORY
			FOR n := 199 TO 0 BY -1 DO
							
				astEventsHistory[n+1].sEventTex				:= astEventsHistory[n].sEventTex;
				astEventsHistory[n+1].sType					:= astEventsHistory[n].sType;
				astEventsHistory[n+1].abType				:= astEventsHistory[n].abType;
				astEventsHistory[n+1].sDate					:= astEventsHistory[n].sDate;										
				astEventsHistory[n+1].sTime					:= astEventsHistory[n].sTime;
				
			END_FOR
			
			astEventsHistory[0].sEventTex				:= stStationEvents[k[0]].aEvents[k[1]].bEventTextHMI;
			astEventsHistory[0].sType					:= 'Cycle Stop Fault';
			astEventsHistory[0].abType					:= 1;
			astEventsHistory[0].sDate					:= 	sSystemTime;										
			astEventsHistory[0].sTime					:= 	sSystemDate;
															
			l											:= l + 1;						
		END_IF
		
		IF stStationEvents[k[0]].aEvents[k[1]].bCycleStopRequest AND stStationEvents[k[0]].aEvents[k[1]].bEventFlag AND NOT stStationEvents[k[0]].aEvents[k[1]].bActive THEN
			
			//ACTIVE EVENTS
			astActiveEvents[l].sEventTex				:= 	stStationEvents[k[0]].aEvents[k[1]].bEventTextHMI;
			astActiveEvents[l].sType					:= 'Cycle Stop Request';						
			astActiveEvents[l].abType					:= 2; 
			astActiveEvents[l].sSolution				:= stStationEvents[k[0]].aEvents[k[1]].sSolution;
			stStationEvents[k[0]].aEvents[k[1]].bActive := TRUE;
			
			//EVENTS HISTORY
			FOR n := 199 TO 0 BY -1 DO
							
				astEventsHistory[n+1].sEventTex				:= astEventsHistory[n].sEventTex;
				astEventsHistory[n+1].sType					:= astEventsHistory[n].sType;
				astEventsHistory[n+1].abType				:= astEventsHistory[n].abType;
				astEventsHistory[n+1].sDate					:= astEventsHistory[n].sDate;										
				astEventsHistory[n+1].sTime					:= astEventsHistory[n].sTime;
				
			END_FOR

			astEventsHistory[0].sEventTex				:= stStationEvents[k[0]].aEvents[k[1]].bEventTextHMI;
			astEventsHistory[0].sType					:= 'Cycle Stop Request';
			astEventsHistory[0].abType					:= 2;
			astEventsHistory[0].sDate					:= 	sSystemTime;										
			astEventsHistory[0].sTime					:= 	sSystemDate;
															
															
			l											:= l + 1;							
		END_IF
		
		IF stStationEvents[k[0]].aEvents[k[1]].bMessage AND stStationEvents[k[0]].aEvents[k[1]].bEventFlag AND NOT stStationEvents[k[0]].aEvents[k[1]].bActive THEN
			
			//ACTIVE EVENTS
			astActiveEvents[l].sEventTex				:= 	stStationEvents[k[0]].aEvents[k[1]].bEventTextHMI;
			astActiveEvents[l].sType					:= 'Message';						
			astActiveEvents[l].abType					:= 3; 
			astActiveEvents[l].sSolution				:= stStationEvents[k[0]].aEvents[k[1]].sSolution;
			stStationEvents[k[0]].aEvents[k[1]].bActive := TRUE;
			
			//EVENTS HISTORY
			FOR n := 199 TO 0 BY -1 DO
							
				astEventsHistory[n+1].sEventTex				:= astEventsHistory[n].sEventTex;
				astEventsHistory[n+1].sType					:= astEventsHistory[n].sType;
				astEventsHistory[n+1].abType				:= astEventsHistory[n].abType;
				astEventsHistory[n+1].sDate					:= astEventsHistory[n].sDate;										
				astEventsHistory[n+1].sTime					:= astEventsHistory[n].sTime;
				
			END_FOR

			astEventsHistory[0].sEventTex				:= stStationEvents[k[0]].aEvents[k[1]].bEventTextHMI;
			astEventsHistory[0].sType					:= 'Message';
			astEventsHistory[0].abType					:= 3;
			astEventsHistory[0].sDate					:= 	sSystemTime;										
			astEventsHistory[0].sTime					:= 	sSystemDate;
															
			l											:= l + 1;
										
		END_IF
		
		
	END_FOR

END_FOR
ELSIF bResetFaults THEN
	FOR l := 0 TO 50 DO
	
			astActiveEvents[l].sEventTex			:= 	'';
			astActiveEvents[l].sType				:= '';						
			astActiveEvents[l].abType				:= 0; 
			astActiveEvents[l].sSolution			:= '';
			
	END_FOR	
	
	FOR k[0] := 0 TO 3 DO
	
		FOR k[1] := 0 TO 100 DO
	
			stStationEvents[k[0]].aEvents[k[1]].bActive	:= FALSE;
		END_FOR
	END_FOR
	
	l												:= 0;
	k[0]											:= 0;
	k[1]											:= 0;	
	bResetFaults									:= FALSE;
ELSE
	
	k[0]											:= 0;
	k[1]											:= 0;
	
END_IF


//



																		//0:Immediate Fault
																		//1:Cycle Stop Fault
																		//2: Cycle Stop Request
																		//3: Message
END_ACTION

ACTION ACT_EventTextAssigment:

FOR j[0] := 0 TO 3 DO
	
	FOR j[1] := 0 TO 100 DO 
		
		IF stStationEvents[j[0]].aEvents[j[1]].bImmediateFault THEN
			
			m[0]											:= m[0]+1;
			
			stStationEvents[j[0]].aEvents[j[1]].bEventTextHMI	:= 		CONCAT( STR1 := 'Immediate Fault N ', STR2 := 
																CONCAT( STR1 := DINT_TO_STRING(m[0]), str2 := 
																CONCAT( STR1 :=' - Station ' , STR2 := 
																CONCAT( STR1 := DINT_TO_STRING(j[0]), STR2 := 
																CONCAT( STR1 :=' - ', str2 := stStationEvents[j[0]].aEvents[j[1]].bEventText )))));
			stStationEvents[j[0]].aEvents[j[1]].bAssignedID	:= 	m[0];				
			
			//EVENTS ASSIGMENT
			stEventsAssigment.astImmediateFaultEvents[m[0]].sEventText	:= stStationEvents[j[0]].aEvents[j[1]].bEventTextHMI;
			stEventsAssigment.astImmediateFaultEvents[m[0]].sSolution	:= stStationEvents[j[0]].aEvents[j[1]].sSolution;
			
		ELSIF stStationEvents[j[0]].aEvents[j[1]].bCycleStopFault THEN
			
			m[1]											:= m[1]+1;
			
			stStationEvents[j[0]].aEvents[j[1]].bEventTextHMI	:= 		CONCAT( STR1 := 'Cycle Stop Fault N ', STR2 := 
																CONCAT( STR1 := DINT_TO_STRING(m[1]), str2 := 
																CONCAT( STR1 :=' - Station ' , STR2 := 
																CONCAT( STR1 := DINT_TO_STRING(j[0]), STR2 := 
																CONCAT( STR1 :=' - ', str2 := stStationEvents[j[0]].aEvents[j[1]].bEventText )))));
			stStationEvents[j[0]].aEvents[j[1]].bAssignedID	:= 	m[1];													
			
			//EVENTS ASSIGMENT
			stEventsAssigment.astCycleStopFaultEvents[m[1]].sEventText	:= stStationEvents[j[0]].aEvents[j[1]].bEventTextHMI;
			stEventsAssigment.astCycleStopFaultEvents[m[1]].sSolution	:= stStationEvents[j[0]].aEvents[j[1]].sSolution;
			
		ELSIF stStationEvents[j[0]].aEvents[j[1]].bCycleStopRequest THEN
		
			m[2]											:= m[2]+1;	
			
			stStationEvents[j[0]].aEvents[j[1]].bEventTextHMI	:= 		CONCAT( STR1 := 'Cycle Stop Request N ', STR2 := 
																CONCAT( STR1 := DINT_TO_STRING(m[2]), str2 := 
																CONCAT( STR1 :=' - Station ' , STR2 := 
																CONCAT( STR1 := DINT_TO_STRING(j[0]), STR2 := 
																CONCAT( STR1 :=' - ', str2 := stStationEvents[j[0]].aEvents[j[1]].bEventText )))));
			stStationEvents[j[0]].aEvents[j[1]].bAssignedID	:= 	m[2];													

			//EVENTS ASSIGMENT
			stEventsAssigment.astCycleStopRequestEvents[m[2]].sEventText	:= stStationEvents[j[0]].aEvents[j[1]].bEventTextHMI;
			stEventsAssigment.astCycleStopRequestEvents[m[2]].sSolution	:= stStationEvents[j[0]].aEvents[j[1]].sSolution;
			
		ELSIF stStationEvents[j[0]].aEvents[j[1]].bMessage THEN
			
			m[3]											:= m[3]+1;
			
			stStationEvents[j[0]].aEvents[j[1]].bEventTextHMI	:= 		CONCAT( STR1 := 'Message N ', STR2 := 
																CONCAT( STR1 := DINT_TO_STRING(m[3]), str2 := 
																CONCAT( STR1 :=' - Station ' , STR2 := 
																CONCAT( STR1 := DINT_TO_STRING(j[0]), STR2 := 
																CONCAT( STR1 :=' - ', str2 := stStationEvents[j[0]].aEvents[j[1]].bEventText )))));
			stStationEvents[j[0]].aEvents[j[1]].bAssignedID	:= 	m[3];													
				
			//EVENTS ASSIGMENT
			stEventsAssigment.astMessage[m[3]].sEventText	:= stStationEvents[j[0]].aEvents[j[1]].bEventTextHMI;
			stEventsAssigment.astMessage[m[3]].sSolution	:= stStationEvents[j[0]].aEvents[j[1]].sSolution;	
			
		END_IF
		
	END_FOR
	
	
END_FOR
j[0]														:= 0;
j[1]														:= 0;
m[0]														:= 0;
m[1]														:= 0;
m[2]														:= 0;
m[3]														:= 0;
END_ACTION

ACTION ACT_FaultTrig:
IF bPulse THEN
	

	FOR i[0] := 0 TO 3 DO
	//IMMEDIATE FAULT
		FOR i[1] :=0 TO 100 DO
			
			//IMMEDIATE FAULT
			IF stStationEvents[i[0]].aEvents[i[1]].bImmediateFault AND stStationEvents[i[0]].aEvents[i[1]].bEventFlag THEN
	
				stStationEvents[i[0]].bImmediateFault						:= TRUE;
		
			ELSIF bResetFaults THEN
				stStationEvents[i[0]].bImmediateFault						:= FALSE;
			END_IF
			//STOP FAULT
			IF stStationEvents[i[0]].aEvents[i[1]].bCycleStopFault AND stStationEvents[i[0]].aEvents[i[1]].bEventFlag THEN
	
				stStationEvents[i[0]].bCycleStopFault						:= TRUE;
		
			ELSIF bResetFaults THEN
				stStationEvents[i[0]].bCycleStopFault						:= FALSE;
			END_IF
		
			//STOP REQUEST
			IF stStationEvents[i[0]].aEvents[i[1]].bCycleStopRequest AND stStationEvents[i[0]].aEvents[i[1]].bEventFlag THEN
	
				stStationEvents[i[0]].bCycleStopRequest						:= TRUE;
		
			ELSIF bResetFaults THEN
				stStationEvents[i[0]].bCycleStopRequest						:= FALSE;
			END_IF
		
		END_FOR
	END_FOR

ELSE 	i[0]														:= 0;
		i[1]														:= 0;	
END_IF
END_ACTION

END_FUNCTION_BLOCK

// ---- POUs/Utilities/FB_UserLog.TcPOU
FUNCTION_BLOCK FB_UserLog
VAR_INPUT
	
	nNumberOfData				: DINT;
	bSaveSignal					: BOOL;
	sUser						: STRING;
	sGroup						: STRING;
	sDate						: STRING;
	sTime						: STRING;

END_VAR
VAR_OUTPUT
	
END_VAR
VAR
	rSaveSignal					: R_TRIG;
	i							: DINT;
END_VAR
VAR_IN_OUT
	
	aDataOutput					: ARRAY [*] OF ST_UserLog;
	
END_VAR

rSaveSignal( CLK := bSaveSignal);

IF rSaveSignal.Q THEN
	
	FOR i := nNumberOfData TO 0 BY -1 DO
		
		aDataOutput[i+1]		:= aDataOutput[i];
		
	END_FOR
	
	aDataOutput[0].sDate		:= sDate;
	aDataOutput[0].sGroup		:= sGroup;
	aDataOutput[0].sTime		:= sTime;
	aDataOutput[0].sUser		:= sUser;
	
END_IF

END_FUNCTION_BLOCK

// ---- POUs/A_MASTER/A_3_PRG_FaultHandling.TcPOU
PROGRAM A_3_PRG_FaultHandling
VAR
	

	bEventsFlag					: ARRAY [0..100] OF BOOL;



END_VAR

a_ACT_Set_Events();
/////////////////////////////////////////////////////////////////////////////////////MASTER FAULT MONITORS////////////////////////////////////////////////////////////////////////////////////


stMasterCtrl.bNoImmediateFault 										:= 	NOT stStationEvents[0].bImmediateFault AND NOT stStationEvents[1].bImmediateFault AND
                                            							NOT stStationEvents[2].bImmediateFault AND NOT stStationEvents[3].bImmediateFault;

stMasterCtrl.bNoCycleStopFault 										:= NOT stStationEvents[0].bCycleStopFault AND NOT stStationEvents[1].bCycleStopFault AND
                          												NOT stStationEvents[2].bCycleStopFault AND NOT stStationEvents[3].bCycleStopFault;

stMasterCtrl.bCycleStopRequest										:= stStationEvents[0].bCycleStopRequest OR stStationEvents[0].bCycleStopRequest OR
																		stStationEvents[0].bCycleStopRequest OR stStationEvents[0].bCycleStopRequest;

ACTION a_ACT_Set_Events:
//IMMEDIATE FAULTS

stStationEvents[0].aEvents[0].bImmediateFault				:= TRUE;
stStationEvents[0].aEvents[0].bEventFlag					:= bEventsFlag[0];
stStationEvents[0].aEvents[0].bEventText					:= 'ST1 EVENT 0';
stStationEvents[0].aEvents[0].sSolution						:= 'Solution 5';


//CYCLE STOP FAULT

stStationEvents[0].aEvents[1].bCycleStopFault				:= TRUE;
stStationEvents[0].aEvents[1].bEventFlag					:= bEventsFlag[1];
stStationEvents[0].aEvents[1].bEventText					:= 'ST1 EVENT 1';
stStationEvents[0].aEvents[1].sSolution						:= 'Solution 6';


//CYCLE STOP REQUEST

stStationEvents[0].aEvents[2].bCycleStopRequest			:= TRUE;
stStationEvents[0].aEvents[2].bEventFlag					:= bEventsFlag[2];
stStationEvents[0].aEvents[2].bEventText					:= 'ST1 EVENT 7';
END_ACTION

END_PROGRAM

// ---- POUs/C_HMI/C_1_PRG_MainHMI.TcPOU
PROGRAM C_1_PRG_MainHMI
VAR
END_VAR

a_ACT_MachineStatusBaner();

ACTION a_ACT_MachineStatusBaner:
//Machine status banner action
//SYSTEM POWER UP
IF stMachineStatus.bSystemPowerUp THEN	
	stStatusBanner.sMachineStatusText 							:= 'SYSTEM POWER UP';	
	stStatusBanner.nMachineStatusColour 						:= nWHITE;
	stStatusBanner.nMachineStatusTxtCol 						:= nBLACK;
	stStatusBanner.sBannerBckColor 								:= sWHITE;
	stStatusBanner.sBannerTextColor 							:= sBLACK;
END_IF

(* IMMEDIATE STOPPED *)
IF stMachineStatus.bImmediateStopped THEN	
	stStatusBanner.sMachineStatusText 							:= 'IMMEDIATE STOPPED';		
	stStatusBanner.nMachineStatusColour 						:= nBLACK;
	stStatusBanner.nMachineStatusTxtCol 						:= nWHITE;
	stStatusBanner.sBannerBckColor 								:= sBLACK;
	stStatusBanner.sBannerTextColor 							:= sWHITE;	
END_IF

(* SYSTEM INITIALISING *)
IF stMachineStatus.bInitialising THEN	
	stStatusBanner.sMachineStatusText 							:= 'SYSTEM INITIALIZING';		
	stStatusBanner.nMachineStatusColour 						:= nYELLOW;
	stStatusBanner.nMachineStatusTxtCol 						:= nBLACK;
	stStatusBanner.sBannerBckColor 								:= sYELLOW;
	stStatusBanner.sBannerTextColor 							:= sBLACK;
END_IF
(*
(* SYSTEM IN STANDBY *)
IF stMachineStatus.bSystemStandby THEN
	stMachineStatus.sMachineStatusText := 'SYSTEM IN STANDBY';
	stMachineStatus.nMachineStatusColour := nORANGE;
	stMachineStatus.nMachineStatusTxtCol := nWHITE;
END_IF
*)
(* SYSTEM READY TO START FLASH ON *)
IF stMachineStatus.bReadyToStart AND stPuls.bFlash1Hz THEN
	stStatusBanner.sMachineStatusText 							:= 'SYSTEM READY TO START';		
	stStatusBanner.nMachineStatusColour 						:= nGREEN;
	stStatusBanner.nMachineStatusTxtCol 						:= nWHITE;
	stStatusBanner.sBannerBckColor 								:= sGREEN;
	stStatusBanner.sBannerTextColor 							:= sWHITE;
ELSIF stMachineStatus.bReadyToStart AND NOT stPuls.bFlash1Hz THEN	
	stStatusBanner.sMachineStatusText 							:= 'SYSTEM READY TO START';		
	stStatusBanner.nMachineStatusColour 						:= nWHITE;
	stStatusBanner.nMachineStatusTxtCol 						:= nGREEN;
	stStatusBanner.sBannerBckColor 								:= sWHITE;
	stStatusBanner.sBannerTextColor 							:= sGREEN;
END_IF

(* SYSTEM AUTO CYCLE *)
IF stMachineStatus.bAutoCycle THEN	
	stStatusBanner.sMachineStatusText 							:= 'SYSTEM AUTO CYCLE';		
	stStatusBanner.nMachineStatusColour 						:= nGREEN;
	stStatusBanner.nMachineStatusTxtCol 						:= nWHITE;
	stStatusBanner.sBannerBckColor 								:= sGREEN;
	stStatusBanner.sBannerTextColor 							:= sWHITE;	
END_IF

(*(* SYSTEM DWELL *)
IF stMachineStatus.THEN	
	GVL_MASTER.stMachineStatus.sMachineStatusText := 'SYSTEM DWELL';		
	GVL_MASTER.stMachineStatus.nMachineStatusColour := nORANGE;
	GVL_MASTER.stMachineStatus.nMachineStatusTxtCol := nWHITE;
	GVL_MASTER.stMachineStatus.sBannerBckColor := sORANGE;
	GVL_MASTER.stMachineStatus.sBannerTextColor := sWHITE;	
END_IF*)

(* STOPPING *)
IF stMachineStatus.bStopping AND stPuls.bFlash1Hz THEN	
	stStatusBanner.sMachineStatusText 							:= 'STOPPING';		
	stStatusBanner.nMachineStatusColour 						:= nBLACK;
	stStatusBanner.nMachineStatusTxtCol 						:= nWHITE;
	stStatusBanner.sBannerBckColor 								:= sBLACK;
	stStatusBanner.sBannerTextColor 							:= sWHITE;	
ELSIF stMachineStatus.bStopping AND NOT stPuls.bFlash1Hz THEN	
	stStatusBanner.sMachineStatusText 							:= 'STOPPING';		
	stStatusBanner.nMachineStatusColour 						:= nWHITE;
	stStatusBanner.nMachineStatusTxtCol 						:= nBLACK;
	stStatusBanner.sBannerBckColor 								:= sWHITE;
	stStatusBanner.sBannerTextColor 							:= sBLACK;	
END_IF

(* CYCLE STOPPED *)
IF stMachineStatus.bCycleStopped THEN	
	stStatusBanner.sMachineStatusText 							:= 'CYCLE STOPPED';		
	stStatusBanner.nMachineStatusColour 						:= nBLACK;
	stStatusBanner.nMachineStatusTxtCol 						:= nWHITE;
	stStatusBanner.sBannerBckColor 								:= sBLACK;
	stStatusBanner.sBannerTextColor 							:= sWHITE;	
END_IF

(* IMMEDIATE FAULT FLASH ON *)
IF stMachineStatus.bImmediateFault AND stPuls.bFlash1Hz THEN	
	stStatusBanner.sMachineStatusText 							:= 'IMMEDIATE FAULT';		
	stStatusBanner.nMachineStatusColour 						:= nRED;
	stStatusBanner.nMachineStatusTxtCol 						:= nWHITE;
	stStatusBanner.sBannerBckColor 								:= sRED;
	stStatusBanner.sBannerTextColor 							:= sWHITE;	
ELSIF stMachineStatus.bImmediateFault AND NOT stPuls.bFlash1Hz THEN	
	stStatusBanner.sMachineStatusText 							:= 'IMMEDIATE FAULT';		
	stStatusBanner.nMachineStatusColour 						:= nWHITE;
	stStatusBanner.nMachineStatusTxtCol 						:= nBLACK;
	stStatusBanner.sBannerBckColor 								:= sWHITE;
	stStatusBanner.sBannerTextColor 							:= sBLACK;	
END_IF

(* CYCLE STOP FAULT FLASH ON *)
IF stMachineStatus.bCycleStopFault AND stPuls.bFlash1Hz THEN	
	stStatusBanner.sMachineStatusText 							:= 'CYCLE STOP FAULT';		
	stStatusBanner.nMachineStatusColour 						:= nRED;
	stStatusBanner.nMachineStatusTxtCol 						:= nWHITE;
	stStatusBanner.sBannerBckColor 								:= sRED;
	stStatusBanner.sBannerTextColor 							:= sWHITE;	
ELSIF GVL_MASTER.stMachineStatus.bCycleStopFault AND NOT stPuls.bFlash1Hz THEN	
	stStatusBanner.sMachineStatusText 							:= 'CYCLE STOP FAULT';		
	stStatusBanner.nMachineStatusColour 						:= nWHITE;
	stStatusBanner.nMachineStatusTxtCol 						:= nRED;
	stStatusBanner.sBannerBckColor 								:= sWHITE;
	stStatusBanner.sBannerTextColor 							:= sRED;	
END_IF

(* MANUAL MODE *)
IF stMachineStatus.bManualMode THEN	
	stStatusBanner.sMachineStatusText 							:= 'MANUAL MODE';		
	stStatusBanner.nMachineStatusColour 						:= nBLUE;
	stStatusBanner.nMachineStatusTxtCol 						:= nWHITE;
	stStatusBanner.sBannerBckColor 								:= sBLUE;
	stStatusBanner.sBannerTextColor 							:= sWHITE;	
END_IF
END_ACTION

END_PROGRAM

// ---- POUs/D_CSV/D_1_WriteDataToCSV.TcPOU
PROGRAM D_1_WriteDataToCSV
VAR
	
	bWrite			: BOOL := FALSE;(* Rising edge starts program execution *)
	sFileName		: T_MaxString ;(* CSV destination file path and name *)
	sCSVLine		: T_MaxString := '';(* Single CSV text line (row, record), we are using string as record buffer (your are able to see created fields) *)
	sCSVField		: T_MaxString := '';(* Single CSV field value (column, record field) *)
	bBusy			: BOOL;
	bError			: BOOL;
	nErrId			: UDINT;
	nRow	 		: UDINT 	:= 0;(* Row number (record) *)
	nColumn			: UDINT 	:= 0;(* Column number (record field) *)
	hFile			: UINT		:= 0;(* File handle of the source file *)
	step			: DWORD 	:= 0;
	fbFileOpen		: FB_FileOpen;(* Opens file *)
	fbFileClose		: FB_FileClose;(* Closes file *)
	fbFilePuts		: FB_FilePuts;(* Writes one record (line) *)
	fbWriter		: FB_CSVMemBufferWriter;(* Helper function block used to create CSV data bytes (single record line) *)

	database		: ARRAY[0..MAX_CSV_ROWS, 0..MAX_CSV_COLUMNS ] OF STRING(MAX_CSV_FIELD_LENGTH);  
	
	nCSVIndex		: DINT;
	sCSVIndex		: STRING;
	rChangeCSVTrigger: R_TRIG;
	i				: DINT;
	j				: DINT;
END_VAR

a_ACT_IO();
b_SettingsToCsv();

CASE step OF
	0:	(* Wait for rising edge at bWrite variable *)
		IF bWrite THEN
			bWrite 	:= FALSE;
			bBusy 	:= TRUE;
			bError	:= FALSE;
			nErrId	:= 0;
			hFile	:= 0;
			nRow	:= 0;
			nColumn	:= 0;
			step 	:= 1;
		END_IF

	1:	(* Open source file *)
		fbFileOpen(  bExecute := FALSE  );
		fbFileOpen( sNetId := NetAmsId , sPathName := sFileName, nMode := FOPEN_MODEWRITE OR FOPEN_MODETEXT,(* Open file in TEXT mode! *)
					ePath := PATH_GENERIC, bExecute := TRUE );
		step := 2;

	2:(* Wait until open not busy *)
		fbFileOpen( bExecute := FALSE, bError => bError, nErrID => nErrID, hFile => hFile );
		IF NOT fbFileOpen.bBusy THEN
			IF NOT fbFileOpen.bError THEN
				step := 3;
			ELSE(* Error: file not found? *)
				step := 100;
			END_IF
		END_IF

	3:(* Convert one PLC record to CSV format *)
		sCSVLine := '';
		fbWriter.eCmd := eEnumCmd_First;(* Write first field value *)
		IF nRow <= MAX_CSV_ROWS THEN

			FOR nColumn := 0 TO MAX_CSV_COLUMNS BY 1 DO

				sCSVField := STRING_TO_CSVFIELD( database[ nRow, nColumn ], FALSE );(* TODO: Get field value from your application *)

				(* Add new field to the record buffer *)
				fbWriter( 	pBuffer := ADR( sCSVLine ), cbBuffer := SIZEOF( sCSVLine ) - 1, putValue := sCSVField, pValue := 0, cbValue := 0,
							bCRLF := ( nColumn = MAX_CSV_COLUMNS ) );(* bCRLF == TRUE => Write CRLF after the last field value *)
				IF fbWriter.bOk THEN
					fbWriter.eCmd := eEnumCmd_Next;(* Write next field value *)
				ELSE(* Error *)
					step := 100;
					RETURN;
				END_IF
				
			END_FOR(* FOR nColumn := 0... *)

			(* FB_FilePuts adds allready CR (carriage return) to the written line.
			We have to replace the $R$L characters with $L character to avoid double CR. *)
			IF RIGHT( sCSVLine, 2 ) = '$R$L' THEN
				sCSVLine := REPLACE( sCSVLine, '$L', 2, LEN( sCSVLine ) - 1 );
			END_IF

			nRow := nRow + 1;(* Increment number of created records (rows) *)
			step := 4;(* Write record to the file *)

		ELSE(* All rows written => Close file *)
			step := 10;
		END_IF

	4:	(* Write single text line *)
		fbFilePuts( bExecute := FALSE );
		fbFilePuts( sNetId := NetAmsId , hFile := hFile, sLine := sCSVLine, bExecute := TRUE );
		step := 5;

	5:(* Wait until write not busy *)
		fbFilePuts( bExecute := FALSE, bError => bError, nErrID => nErrID );
		IF NOT fbFilePuts.bBusy THEN
			IF NOT fbFilePuts.bError THEN
				step := 3;(* Write next record *)
			ELSE(* Error *)
				step := 100;
			END_IF
		END_IF

	10:	(* Close source file *)
		fbFileClose( bExecute := FALSE );
		fbFileClose( sNetId := NetAmsId , hFile := hFile, bExecute := TRUE );
		step := 11;

	11:(* Wait until close not busy *)
		fbFileClose( bExecute := FALSE, bError => bError, nErrID => nErrID );
		IF ( NOT fbFileClose.bBusy ) THEN
			hFile := 0;
			step := 100;
		END_IF

	100: (* Error or ready step => cleanup *)
		IF ( hFile <> 0 ) THEN
			step := 10; (* Close the source file *)
		ELSE
			bBusy := FALSE;
			step := 0;	(* Ready *)
		END_IF

END_CASE

ACTION a_ACT_IO:
//database	:=

//INPUTS
bWrite									:= stCSVProcess.bWriteData;

//OUTPUTS
stCSVProcess.bBusy						:= bBusy;
stCSVProcess.bError						:= bError;
END_ACTION

ACTION b_SettingsToCsv:
rChangeCSVTrigger( CLK := nIndexDataHistory = 200);
IF nIndexDataHistory = 200 THEN
	FOR i := 0 TO 200 DO
		FOR j := 0 TO 28 DO
			database[i,j]				:='';
		END_FOR
	END_FOR 
END_IF
IF rChangeCSVTrigger.Q THEN
	nCSVIndex							:= nCSVIndex + 1;
	nIndexDataHistory 					:= 0;
END_IF

sCSVIndex 								:= DINT_TO_STRING(nCSVIndex);

sFileName 								:= CONCAT(stCSVProcess.sFileName1,CONCAT(sCSVIndex,stCSVProcess.sFileName2));

IF nCSVIndex = 100 THEN
	nCSVIndex 							:= 0;
END_IF

database[nIndexDataHistory,0]			:= aDataHistory[0].sSetting1_1;	
database[nIndexDataHistory,1]			:= DINT_TO_STRING(aDataHistory[0].nSetting2_1);

IF 	aDataHistory[0].bSetting3_1 THEN
	database[nIndexDataHistory,2]			:= 'TRUE';	
ELSE database[nIndexDataHistory,2]			:= 'FALSE';
END_IF
	
database[nIndexDataHistory,3]			:= aDataHistory[0].sDATA1_1;	
database[nIndexDataHistory,4]			:= DINT_TO_STRING(aDataHistory[0].nDATA2_1);	

IF 	aDataHistory[0].bDATA3_1 THEN
	database[nIndexDataHistory,5]			:= 'TRUE';	
ELSE database[nIndexDataHistory,5]			:= 'FALSE';
END_IF
	
IF 	aDataHistory[0].bPass_1 THEN
	database[nIndexDataHistory,6]			:= 'TRUE';	
ELSE database[nIndexDataHistory,6]			:= '';
END_IF

IF 	aDataHistory[0].bFail_1 THEN
	database[nIndexDataHistory,7]			:= 'TRUE';	
ELSE database[nIndexDataHistory,7]			:= '';
END_IF
	
database[nIndexDataHistory,8]			:= aDataHistory[0].sSetting1_2;
database[nIndexDataHistory,9]			:= DINT_TO_STRING(aDataHistory[0].nSetting2_2);	

IF 	aDataHistory[0].bSetting3_2 THEN
	database[nIndexDataHistory,10]			:= 'TRUE';	
ELSE database[nIndexDataHistory,10]			:= 'FALSE';
END_IF
	
database[nIndexDataHistory,11]			:= aDataHistory[0].sDATA1_2;	
database[nIndexDataHistory,12]			:= DINT_TO_STRING(aDataHistory[0].nDATA2_2);	

IF 	aDataHistory[0].bDATA3_2 THEN
	database[nIndexDataHistory,13]			:= 'TRUE';	
ELSE database[nIndexDataHistory,13]			:= 'FALSE';
END_IF
	
IF 	aDataHistory[0].bPass_2 THEN
	database[nIndexDataHistory,14]			:= 'TRUE';	
ELSE database[nIndexDataHistory,14]			:= '';
END_IF

IF 	aDataHistory[0].bFail_2 THEN
	database[nIndexDataHistory,15]			:= 'TRUE';	
ELSE database[nIndexDataHistory,15]			:= '';
END_IF
	
database[nIndexDataHistory,16]			:= aDataHistory[0].sSetting1_3;
database[nIndexDataHistory,17]			:= DINT_TO_STRING(aDataHistory[0].nSetting2_3);	

IF 	aDataHistory[0].bSetting3_3 THEN
	database[nIndexDataHistory,18]			:= 'TRUE';	
ELSE database[nIndexDataHistory,18]			:= 'FALSE';
END_IF
	
database[nIndexDataHistory,19]			:= aDataHistory[0].sDATA1_3;	
database[nIndexDataHistory,20]			:= DINT_TO_STRING(aDataHistory[0].nDATA2_3);

IF 	aDataHistory[0].bDATA3_3 THEN
	database[nIndexDataHistory,21]			:= 'TRUE';	
ELSE database[nIndexDataHistory,21]			:= 'FALSE';
END_IF	
	
IF 	aDataHistory[0].bPass_3 THEN
	database[nIndexDataHistory,22]			:= 'TRUE';	
ELSE database[nIndexDataHistory,22]			:= '';
END_IF

IF 	aDataHistory[0].bFail_3 THEN
	database[nIndexDataHistory,23]			:= 'TRUE';	
ELSE database[nIndexDataHistory,23]			:= '';
END_IF
	
IF 	aDataHistory[0].bPass THEN
	database[nIndexDataHistory,24]			:= 'TRUE';	
ELSE database[nIndexDataHistory,24]			:= '';
END_IF

IF 	aDataHistory[0].bFail THEN
	database[nIndexDataHistory,25]			:= 'TRUE';	
ELSE database[nIndexDataHistory,25]			:= '';
END_IF

		
database[nIndexDataHistory,26]			:= aDataHistory[0].sData;		
database[nIndexDataHistory,27]			:= aDataHistory[0].sTime;
END_ACTION

END_PROGRAM

// ---- POUs/A_MASTER/A_4_PRG_MasterSystemTime.TcPOU
PROGRAM A_4_PRG_MasterSystemTime
VAR

END_VAR

END_PROGRAM

// ---- POUs/B_STATIONS/B_1_STATION_1/B_1_1_PRG_Master_Station_1.TcPOU
PROGRAM B_1_1_PRG_Master_Station_1

VAR
	eState								: E_Station1_State;
	tonErrorReset						: TON;
	tonStationStopped					: TON;
	ctuErrorCounter						: CTU;
	rGoodStatistics						: R_TRIG;
	rBadStatistics						: R_TRIG;
	rEfficency							: STRING(510);
	
	bPersistentError					: BOOL;
	
	bEventsFlag							: ARRAY [0..100] OF BOOL;
/////////////////////////////////////////////////////////////////////////////////////I O/////////////////////////////////////////////////////////////////////////////////////	
	bStopped							: BOOL;
	bError								: BOOL;
	bReady								: BOOL;
	bDone								: BOOL;
	bPass								: BOOL;
	bFail								: BOOL;

	
END_VAR

VAR_INPUT	
	
	CMD									:ST_StationCMD;	
	
END_VAR

VAR_OUTPUT	
	
	STATUS								:ST_StationStatus;	
	
END_VAR

a_ACT_Ctrl_Station_1();
b_ACT_IO();
c_ACT_Statistics_Station_1();
d_ACT_Set_Events_Station_1();

ACTION a_ACT_Ctrl_Station_1:
/////////////////////////////////////////////////////////////////////////////////////UTILITIES/////////////////////////////////////////////////////////////////////////////////////
tonErrorReset( IN := (eState = E_Station1_State.RESET_ERROR), PT := T#500MS);
tonStationStopped( IN := bStopped, PT := T#1S);

ctuErrorCounter( CU := eState = E_Station1_State.RESET_ERROR, RESET := ((ctuErrorCounter.CV = 5) AND eState = E_Station1_State.PERSISTENT_ERROR), PV := 5, Q => bPersistentError);



/////////////////////////////////////////////////////////////////////////////////////CONDITIONS/////////////////////////////////////////////////////////////////////////////////////

IF (CMD.bAbort OR bError) AND ( eState			= E_Station1_State.HOMING OR
								eState			= E_Station1_State.READY OR
								eState			= E_Station1_State.MOVEMENT_A OR
								eState			= E_Station1_State.MOVEMENT_B OR
								eState			= E_Station1_State.MOVEMENT_C OR
								eState			= E_Station1_State.READY OR
								eState			= E_Station1_State.DONE) THEN
								
	eState						:= E_Station1_State.STOPPING;
	
END_IF



CASE eState OF
	
	E_Station1_State.ABORTED:
								IF CMD.bEnable AND NOT bError THEN
									eState						:= E_Station1_State.HOMING;
								ELSIF bError THEN
									eState						:= E_Station1_State.ERROR;
								END_IF
	
	E_Station1_State.HOMING:
								IF bReady THEN
									eState						:= E_Station1_State.RESET;
								END_IF
																
	E_Station1_State.RESET:
								stCycleDataStation1.bPass	:= FALSE;
								stCycleDataStation1.bFail	:= FALSE;
								
								eState						:= E_Station1_State.READY;
	E_Station1_State.READY:
								IF CMD.bExecute AND stStation1.Mov1 THEN
									eState						:= E_Station1_State.MOVEMENT_A;
								ELSIF CMD.bExecute AND stStation1.Mov2 THEN
									eState						:= E_Station1_State.MOVEMENT_B;
								ELSIF CMD.bExecute AND stStation1.Mov3 THEN
									eState						:= E_Station1_State.MOVEMENT_C;
								END_IF
	
	E_Station1_State.MOVEMENT_A:
								IF bDone AND stStation1.Mov1 THEN
									eState						:= E_Station1_State.DONE;
								END_IF
	
	E_Station1_State.MOVEMENT_B:
								IF bDone AND stStation1.Mov2 THEN
									eState						:= E_Station1_State.DONE;
								END_IF
	E_Station1_State.MOVEMENT_C:
								IF bDone AND stStation1.Mov3 THEN
									eState						:= E_Station1_State.DONE;
								END_IF
	E_Station1_State.DONE:
								IF  CMD.bReady THEN
									eState						:= E_Station1_State.RESULTS;
								END_IF	
								
	E_Station1_State.RESULTS:
								
								IF bPass THEN
									stCycleDataStation1.bPass	:= TRUE;
								ELSIF bFail THEN
								 	stCycleDataStation1.bFail	:= TRUE;
								END_IF
								
								IF  CMD.bEndCycle THEN
									eState						:= E_Station1_State.RESET;
								END_IF
								
/////////////////////////////////////////////////////////////////////////////////////RESET CMD/////////////////////////////////////////////////////////////////////////////////////			
	
	E_Station1_State.STOPPING: 
								IF tonStationStopped.Q THEN
									IF bError THEN
										eState						:= E_Station1_State.ERROR;
									ELSE eState						:= E_Station1_State.ABORTED;
									END_IF

								END_IF
	
	E_Station1_State.ERROR:
								IF NOT bError THEN
									eState						:= E_Station1_State.ABORTED;
								ELSE eState						:= E_Station1_State.RESET_ERROR;
								END_IF
	
	E_Station1_State.RESET_ERROR:
								IF tonErrorReset.Q AND NOT bPersistentError THEN
									eState						:= E_Station1_State.ERROR;
								ELSIF bPersistentError THEN
									eState						:= E_Station1_State.PERSISTENT_ERROR;
								END_IF
	
	E_Station1_State.PERSISTENT_ERROR:
								IF CMD.bReset THEN
									eState						:= E_Station1_State.ERROR;
								END_IF
	


							
						
								
													
								

ELSE eState := E_Station1_State.ABORTED;
	
END_CASE
/////////////////////////////////////////////////////////////////////////////////////STATUS/////////////////////////////////////////////////////////////////////////////////////

Status.bBusy				:= 	eState			= E_Station1_State.HOMING OR
								eState			= E_Station1_State.MOVEMENT_A OR
								eState			= E_Station1_State.MOVEMENT_B OR
								eState			= E_Station1_State.MOVEMENT_C OR
								eState			= E_Station1_State.STOPPING;
								
Status.bDone				:=	eState			= E_Station1_State.DONE;
											
Status.bError				:= 	(eState			= E_Station1_State.ERROR) OR 
								(eState			= E_Station1_State.RESET_ERROR) OR
								(eState			= E_Station1_State.PERSISTENT_ERROR);
								
Status.bReady				:= 	eState			= E_Station1_State.READY;

Status.bStopped				:= 	eState			= E_Station1_State.ABORTED OR
								eState			= E_Station1_State.READY OR
								eState			= E_Station1_State.ERROR OR
								eState			= E_Station1_State.RESET_ERROR;
END_ACTION

ACTION b_ACT_IO:
//bStopped								:=;
//bError								:=;
//bReady								:=;
//bDone
END_ACTION

ACTION c_ACT_Statistics_Station_1:
stStatisticsHMI[1].sName			:= 'Station 1';


rGoodStatistics( CLK := (stCycleDataStation1.bPass AND (eState = E_Station1_State.RESULTS)) OR bStatisticsTest[0]);
rBadStatistics( CLK := (stCycleDataStation1.bFail AND (eState = E_Station1_State.RESULTS)) OR bStatisticsTest[1]);

IF 	rGoodStatistics.Q THEN
	
	stStatisticsHMI[1].nGood		:= stStatisticsHMI[1].nGood + 1;
	stStatisticsHMI[1].nTotalGood	:= stStatisticsHMI[1].nTotalGood + 1;
	
END_IF
								
IF 	rBadStatistics.Q THEN
	
	stStatisticsHMI[1].nBad			:= stStatisticsHMI[1].nBad + 1;
	stStatisticsHMI[1].nTotalBad	:= stStatisticsHMI[1].nTotalBad + 1;
	
END_IF

IF stStatisticsHMI[1].bResetGood THEN
	stStatisticsHMI[1].nGood		:= 0;
END_IF

IF stStatisticsHMI[1].bResetBad THEN
	stStatisticsHMI[1].nBad			:= 0;
END_IF



IF (( stStatisticsHMI[1].nGood + stStatisticsHMI[1].nBad) <> 0) THEN
	
	rEfficency							:= LREAL_TO_FMTSTR(in := (DINT_TO_REAL(stStatisticsHMI[1].nGood) /( DINT_TO_REAL(stStatisticsHMI[1].nGood) + DINT_TO_REAL(stStatisticsHMI[1].nBad))) * 100.0,iPrecision := 2, bRound := TRUE);
	stStatisticsHMI[1].nEfficency		:= CONCAT(STR1 := '%', STR2 := (rEfficency));

ELSE stStatisticsHMI[1].nEfficency		:= CONCAT(STR1 := '%', STR2 := (DINT_TO_STRING(0)));
	
END_IF
END_ACTION

ACTION d_ACT_Set_Events_Station_1:
//IMMEDIATE FAULTS

stStationEvents[1].aEvents[0].bImmediateFault				:= TRUE;
stStationEvents[1].aEvents[0].bEventFlag					:= bEventsFlag[0];
stStationEvents[1].aEvents[0].bEventText					:= 'ST1 EVENT 0';
stStationEvents[1].aEvents[0].sSolution						:= 'Solution 1';


//CYCLE STOP FAULT

stStationEvents[1].aEvents[1].bCycleStopFault				:= TRUE;
stStationEvents[1].aEvents[1].bEventFlag					:= bEventsFlag[1];
stStationEvents[1].aEvents[1].bEventText					:= 'ST1 EVENT 1';
stStationEvents[1].aEvents[1].sSolution						:= 'Solution 2';


//CYCLE STOP REQUEST

stStationEvents[1].aEvents[2].bCycleStopRequest			:= TRUE;
stStationEvents[1].aEvents[2].bEventFlag					:= bEventsFlag[2];
stStationEvents[1].aEvents[2].bEventText					:= 'ST1 EVENT 2';
stStationEvents[1].aEvents[2].sSolution						:= '';

//Message

stStationEvents[1].aEvents[3].bMessage						:= TRUE;
stStationEvents[1].aEvents[3].bEventFlag					:= bEventsFlag[3];
stStationEvents[1].aEvents[3].bEventText					:= 'Message 3';
stStationEvents[1].aEvents[3].sSolution						:= '';
END_ACTION

END_PROGRAM

// ---- POUs/B_STATIONS/B_2_STATION_2/B_2_1_PRG_Master_Station_2.TcPOU
PROGRAM B_2_1_PRG_Master_Station_2

VAR
	eState								: E_Station2_State;
	tonErrorReset						: TON;
	tonStationStopped					: TON;
	ctuErrorCounter						: CTU;
	rGoodStatistics						: R_TRIG;
	rBadStatistics						: R_TRIG;
	rEfficency							: STRING(510);
	
	bPersistentError					: bool;
/////////////////////////////////////////////////////////////////////////////////////I O/////////////////////////////////////////////////////////////////////////////////////	
	bStopped							: BOOL;
	bError								: BOOL;
	bReady								: BOOL;
	bDone								: BOOL;
	bPass								: BOOL;
	bFail								: BOOL;

	
END_VAR

VAR_INPUT	
	
	CMD									:ST_StationCMD;	
	
END_VAR

VAR_OUTPUT	
	
	STATUS								:ST_StationStatus;	
	
END_VAR

B_2_2_PRG_Fault_Station_2( aAlarms := stAlarms );
a_ACT_Ctrl_Station_2();
b_ACT_IO();
c_ACT_Statistics_Station_2();

ACTION a_ACT_Ctrl_Station_2:
/////////////////////////////////////////////////////////////////////////////////////UTILITIES/////////////////////////////////////////////////////////////////////////////////////
tonErrorReset( IN := (eState = E_Station2_State.RESET_ERROR), PT := T#500MS);
tonStationStopped( IN := bStopped, PT := T#1S);
ctuErrorCounter( CU := eState = E_Station2_State.RESET_ERROR, RESET := ((ctuErrorCounter.CV = 5) AND eState = E_Station2_State.PERSISTENT_ERROR), PV := 5, Q => bPersistentError);

/////////////////////////////////////////////////////////////////////////////////////CONDITIONS/////////////////////////////////////////////////////////////////////////////////////

IF (CMD.bAbort OR bError) AND ( eState			= E_Station2_State.HOMING OR
								eState			= E_Station2_State.READY OR
								eState			= E_Station2_State.MOVEMENT_A OR
								eState			= E_Station2_State.MOVEMENT_B OR
								eState			= E_Station2_State.MOVEMENT_C OR
								eState			= E_Station2_State.READY  OR
								eState			= E_Station2_State.DONE) THEN
								
	eState						:= E_Station2_State.STOPPING;
	
END_IF

CASE eState OF
	
	E_Station2_State.ABORTED:
								IF CMD.bEnable AND NOT bError THEN
									eState						:= E_Station2_State.HOMING;
								ELSIF bError THEN
									eState						:= E_Station2_State.ERROR;
								END_IF
	
	E_Station2_State.HOMING:
								IF bReady THEN
									eState						:= E_Station2_State.READY;
								END_IF
	E_Station1_State.RESET:
								stCycleDataStation2.bPass	:= FALSE;
								stCycleDataStation2.bFail	:= FALSE;
								
								eState						:= E_Station2_State.READY;
	E_Station2_State.READY:
								IF CMD.bExecute AND stStation2.Mov1 THEN
									eState						:= E_Station2_State.MOVEMENT_A;
								ELSIF CMD.bExecute AND stStation2.Mov2 THEN
									eState						:= E_Station2_State.MOVEMENT_B;
								ELSIF CMD.bExecute AND stStation2.Mov3 THEN
									eState						:= E_Station2_State.MOVEMENT_C;
								END_IF
	
	E_Station2_State.MOVEMENT_A:
								IF bDone AND stStation2.Mov1 THEN
									eState						:= E_Station2_State.DONE;
								END_IF
	
	E_Station2_State.MOVEMENT_B:
								IF bDone AND stStation2.Mov2 THEN
									eState						:= E_Station2_State.DONE;
								END_IF
	E_Station2_State.MOVEMENT_C:
								IF bDone AND stStation2.Mov3 THEN
									eState						:= E_Station2_State.DONE;
								END_IF
	E_Station2_State.DONE:
								IF  CMD.bReady THEN
									eState						:= E_Station2_State.READY;
								END_IF	
	E_Station1_State.RESULTS:
								
								IF bPass THEN
									stCycleDataStation2.bPass	:= TRUE;
								ELSIF bFail THEN
								 	stCycleDataStation2.bFail	:= TRUE;
								END_IF
								
								IF  CMD.bEndCycle THEN
									eState						:= E_Station2_State.RESET;
								END_IF
/////////////////////////////////////////////////////////////////////////////////////RESET CMD/////////////////////////////////////////////////////////////////////////////////////

	E_Station2_State.STOPPING: 
								IF tonStationStopped.Q THEN
									IF bError THEN
										eState						:= E_Station2_State.ERROR;
									ELSE eState						:= E_Station2_State.ABORTED;
									END_IF

								END_IF
	
	E_Station2_State.ERROR:
								IF NOT bError THEN
									eState						:= E_Station2_State.ABORTED;
								ELSE eState						:= E_Station2_State.RESET_ERROR;
								END_IF
	
	E_Station2_State.RESET_ERROR:
								IF tonErrorReset.Q AND NOT bPersistentError THEN
									eState						:= E_Station2_State.ERROR;
								ELSIF bPersistentError THEN
									eState						:= E_Station2_State.PERSISTENT_ERROR;
								END_IF
	
	E_Station2_State.PERSISTENT_ERROR:
								IF CMD.bReset THEN
									eState						:= E_Station2_State.ERROR;
								END_IF
								
								

ELSE eState := E_Station2_State.ABORTED;
	
END_CASE
/////////////////////////////////////////////////////////////////////////////////////STATUS/////////////////////////////////////////////////////////////////////////////////////

Status.bBusy				:= 	eState			= E_Station2_State.HOMING OR
								eState			= E_Station2_State.MOVEMENT_A OR
								eState			= E_Station2_State.MOVEMENT_B OR
								eState			= E_Station2_State.MOVEMENT_C OR
								eState			= E_Station2_State.STOPPING;
								
Status.bDone				:=	eState			= E_Station2_State.DONE;
											
Status.bError				:= 	eState			= (E_Station2_State.ERROR OR  E_Station2_State.RESET_ERROR OR E_Station2_State.PERSISTENT_ERROR);

Status.bReady				:= 	eState			= E_Station2_State.READY;

Status.bStopped				:= 	eState			= E_Station2_State.ABORTED OR
								eState			= E_Station2_State.READY OR
								eState			= E_Station2_State.ERROR OR
								eState			= E_Station2_State.RESET_ERROR;
END_ACTION

ACTION b_ACT_IO:
//bStopped								:=;
//bError								:=;
//bReady								:=;
//bDone
END_ACTION

ACTION c_ACT_Statistics_Station_2:
stStatisticsHMI[2].sName			:= 'Station 2';


rGoodStatistics( CLK := (stCycleDataStation2.bPass AND (eState = E_Station2_State.RESULTS)) OR bStatisticsTest[2]);
rBadStatistics( CLK := (stCycleDataStation2.bFail AND (eState = E_Station2_State.RESULTS)) OR bStatisticsTest[3]);

IF 	rGoodStatistics.Q THEN
	
	stStatisticsHMI[2].nGood		:= stStatisticsHMI[2].nGood + 1;
	stStatisticsHMI[2].nTotalGood	:= stStatisticsHMI[2].nTotalGood + 1;
	
END_IF
								
IF 	rBadStatistics.Q THEN
	
	stStatisticsHMI[2].nBad			:= stStatisticsHMI[2].nBad + 1;
	stStatisticsHMI[2].nTotalBad	:= stStatisticsHMI[2].nTotalBad + 1;
	
END_IF

IF stStatisticsHMI[2].bResetGood THEN
	stStatisticsHMI[2].nGood		:= 0;
END_IF

IF stStatisticsHMI[2].bResetBad THEN
	stStatisticsHMI[2].nBad			:= 0;
END_IF

IF (( stStatisticsHMI[2].nGood + stStatisticsHMI[2].nBad) <> 0) THEN
	
	rEfficency							:= LREAL_TO_FMTSTR(in := (DINT_TO_REAL(stStatisticsHMI[2].nGood) /( DINT_TO_REAL(stStatisticsHMI[2].nGood) + DINT_TO_REAL(stStatisticsHMI[2].nBad))) * 100.0,iPrecision := 2, bRound := TRUE);
	stStatisticsHMI[2].nEfficency		:= CONCAT(STR1 := '%', STR2 := (rEfficency));

ELSE stStatisticsHMI[2].nEfficency		:= CONCAT(STR1 := '%', STR2 := (DINT_TO_STRING(0)));
	
END_IF
END_ACTION

END_PROGRAM

// ---- POUs/B_STATIONS/B_3_STATION_3/B_3_1_PRG_Master_Station_3.TcPOU
PROGRAM B_3_1_PRG_Master_Station_3

VAR
	eState								: E_Station2_State;
	tonErrorReset						: TON;
	tonStationStopped					: TON;
	ctuErrorCounter						: CTU;
	rGoodStatistics						: R_TRIG;
	rBadStatistics						: R_TRIG;
	rEfficency							: STRING(510);
	
	bPersistentError					: BOOL;
	bEventsFlag							: ARRAY [0..100] OF BOOL;
/////////////////////////////////////////////////////////////////////////////////////I O/////////////////////////////////////////////////////////////////////////////////////	
	bStopped							: BOOL;
	bError								: BOOL;
	bReady								: BOOL;
	bDone								: BOOL;
	bPass								: BOOL;
	bFail								: BOOL;
	
END_VAR

VAR_INPUT	
	
	CMD									:ST_StationCMD;	
	
END_VAR

VAR_OUTPUT	
	
	STATUS								:ST_StationStatus;	
	
END_VAR

d_ACT_Set_Events_Station_3();
a_ACT_Ctrl_Station_3();
b_ACT_IO();
c_ACT_Statistics_Station_3();

ACTION a_ACT_Ctrl_Station_3:
/////////////////////////////////////////////////////////////////////////////////////UTILITIES/////////////////////////////////////////////////////////////////////////////////////
tonErrorReset( IN := (eState = E_Station3_State.RESET_ERROR), PT := T#500MS);
tonStationStopped( IN := bStopped, PT := T#1S);
ctuErrorCounter( CU := eState = E_Station3_State.RESET_ERROR, RESET := ((ctuErrorCounter.CV = 5) AND eState = E_Station3_State.PERSISTENT_ERROR), PV := 5, Q => bPersistentError);

/////////////////////////////////////////////////////////////////////////////////////CONDITIONS/////////////////////////////////////////////////////////////////////////////////////

IF (CMD.bAbort OR bError) AND ( eState			= E_Station3_State.HOMING OR
								eState			= E_Station3_State.READY OR
								eState			= E_Station3_State.MOVEMENT_A OR
								eState			= E_Station3_State.MOVEMENT_B OR
								eState			= E_Station3_State.MOVEMENT_C OR
								eState			= E_Station3_State.READY OR
								eState			= E_Station3_State.DONE) THEN
								
	eState						:= E_Station3_State.STOPPING;
	
END_IF

IF CMD.bAbort OR NOT CMD.bEnable THEN
	eState						:= E_Station3_State.ABORTED;
END_IF

CASE eState OF
	
	E_Station3_State.ABORTED:
								IF CMD.bEnable AND NOT bError THEN
									eState						:= E_Station3_State.HOMING;
								ELSIF bError THEN
									eState						:= E_Station3_State.ERROR;
								END_IF
	
	E_Station3_State.HOMING:
								IF bReady THEN
									eState						:= E_Station3_State.READY;
								END_IF
	E_Station1_State.RESET:
								stCycleDataStation3.bPass	:= FALSE;
								stCycleDataStation3.bFail	:= FALSE;
								
								eState						:= E_Station3_State.READY;	
	E_Station3_State.READY:
								IF CMD.bExecute AND stStation3.Mov1 THEN
									eState						:= E_Station3_State.MOVEMENT_A;
								ELSIF CMD.bExecute AND stStation3.Mov2 THEN
									eState						:= E_Station3_State.MOVEMENT_B;
								ELSIF CMD.bExecute AND stStation3.Mov3 THEN
									eState						:= E_Station3_State.MOVEMENT_C;
								END_IF
	
	E_Station3_State.MOVEMENT_A:
								IF bDone AND stStation3.Mov1 THEN
									eState						:= E_Station3_State.DONE;
								END_IF
	
	E_Station3_State.MOVEMENT_B:
								IF bDone AND stStation3.Mov2 THEN
									eState						:= E_Station3_State.DONE;
								END_IF
	E_Station3_State.MOVEMENT_C:
								IF bDone AND stStation3.Mov3 THEN
									eState						:= E_Station3_State.DONE;
								END_IF
	E_Station3_State.DONE:
								IF  CMD.bReady THEN
									eState						:= E_Station3_State.READY;
								END_IF
								
	E_Station1_State.RESULTS:
								
								IF bPass THEN
									stCycleDataStation3.bPass	:= TRUE;
								ELSIF bFail THEN
								 	stCycleDataStation3.bFail	:= TRUE;
								END_IF
								
								IF  CMD.bEndCycle THEN
									eState						:= E_Station3_State.RESET;
								END_IF
	/////////////////////////////////////////////////////////////////////////////////////RESET CMD/////////////////////////////////////////////////////////////////////////////////////
	
	E_Station3_State.STOPPING: 
								IF tonStationStopped.Q THEN
									IF bError THEN
										eState						:= E_Station3_State.ERROR;
									ELSE eState						:= E_Station3_State.ABORTED;
									END_IF

								END_IF
	
	E_Station3_State.ERROR:
								IF NOT bError THEN
									eState						:= E_Station3_State.ABORTED;
								ELSE eState						:= E_Station3_State.RESET_ERROR;
								END_IF
	
	E_Station3_State.RESET_ERROR:
								IF tonErrorReset.Q AND NOT bPersistentError THEN
									eState						:= E_Station3_State.ERROR;
								ELSIF bPersistentError THEN
									eState						:= E_Station3_State.PERSISTENT_ERROR;
								END_IF
	
	E_Station3_State.PERSISTENT_ERROR:
								IF CMD.bReset THEN
									eState						:= E_Station3_State.ERROR;
								END_IF
								
								

ELSE eState := E_Station3_State.ABORTED;
	
END_CASE
/////////////////////////////////////////////////////////////////////////////////////STATUS/////////////////////////////////////////////////////////////////////////////////////

Status.bBusy				:= 	eState			= E_Station3_State.HOMING OR
								eState			= E_Station3_State.MOVEMENT_A OR
								eState			= E_Station3_State.MOVEMENT_B OR
								eState			= E_Station3_State.MOVEMENT_C OR
								eState			= E_Station3_State.STOPPING;
								
Status.bDone				:=	eState			= E_Station3_State.DONE;
											
Status.bError				:= 	eState			= (E_Station3_State.ERROR OR  E_Station3_State.RESET_ERROR OR E_Station3_State.PERSISTENT_ERROR);

Status.bReady				:= 	eState			= E_Station3_State.READY;

Status.bStopped				:= 	eState			= E_Station3_State.ABORTED OR
								eState			= E_Station3_State.READY OR
								eState			= E_Station3_State.ERROR OR
								eState			= E_Station3_State.RESET_ERROR;
END_ACTION

ACTION b_ACT_IO:
//bStopped								:=;
//bError								:=;
//bReady								:=;
//bDone
END_ACTION

ACTION c_ACT_Statistics_Station_3:
stStatisticsHMI[3].sName			:= 'Station 3';


rGoodStatistics( CLK := (stCycleDataStation3.bPass AND (eState = E_Station3_State.RESULTS)) OR bStatisticsTest[4]);
rBadStatistics( CLK := (stCycleDataStation3.bFail AND (eState = E_Station3_State.RESULTS)) OR bStatisticsTest[5]);

IF 	rGoodStatistics.Q THEN
	
	stStatisticsHMI[3].nGood		:= stStatisticsHMI[3].nGood + 1;
	stStatisticsHMI[3].nTotalGood	:= stStatisticsHMI[3].nTotalGood + 1;
	
END_IF
								
IF 	rBadStatistics.Q THEN
	
	stStatisticsHMI[3].nBad			:= stStatisticsHMI[3].nBad + 1;
	stStatisticsHMI[3].nTotalBad	:= stStatisticsHMI[3].nTotalBad + 1;
	
END_IF

IF stStatisticsHMI[3].bResetGood THEN
	stStatisticsHMI[3].nGood		:= 0;
END_IF

IF stStatisticsHMI[3].bResetBad THEN
	stStatisticsHMI[3].nBad			:= 0;
END_IF

IF (( stStatisticsHMI[3].nGood + stStatisticsHMI[3].nBad) <> 0) THEN
	
	rEfficency							:= LREAL_TO_FMTSTR(in := (DINT_TO_REAL(stStatisticsHMI[3].nGood) /( DINT_TO_REAL(stStatisticsHMI[3].nGood) + DINT_TO_REAL(stStatisticsHMI[3].nBad))) * 100.0,iPrecision := 2, bRound := TRUE);
	stStatisticsHMI[3].nEfficency		:= CONCAT(STR1 := '%', STR2 := (rEfficency));

ELSE stStatisticsHMI[3].nEfficency		:= CONCAT(STR1 := '%', STR2 := (DINT_TO_STRING(0)));
	
END_IF
END_ACTION

ACTION d_ACT_Set_Events_Station_3:
//IMMEDIATE FAULTS

stStationEvents[3].aEvents[0].bImmediateFault				:= TRUE;
stStationEvents[3].aEvents[0].bEventFlag					:= bEventsFlag[0];
stStationEvents[3].aEvents[0].bEventText					:= 'ST1 EVENT 0';
stStationEvents[3].aEvents[0].sSolution						:= 'Solution 5';


//CYCLE STOP FAULT

stStationEvents[3].aEvents[1].bCycleStopFault				:= TRUE;
stStationEvents[3].aEvents[1].bEventFlag					:= bEventsFlag[1];
stStationEvents[3].aEvents[1].bEventText					:= 'ST1 EVENT 1';
stStationEvents[3].aEvents[1].sSolution						:= 'Solution 6';


//CYCLE STOP REQUEST

stStationEvents[3].aEvents[2].bCycleStopRequest			:= TRUE;
stStationEvents[3].aEvents[2].bEventFlag					:= bEventsFlag[2];
stStationEvents[3].aEvents[2].bEventText					:= 'ST1 EVENT 7';
END_ACTION

END_PROGRAM

// ---- POUs/A_MASTER/A_2_PRG_MachineCtrl.TcPOU
PROGRAM A_2_PRG_MachineCtrl
VAR
/////////////////////////////////////////////////////////////////////////////////////TIMERS & TRIGGERS/////////////////////////////////////////////////////////////////////////////////////

	tonSys_Init					: Tc2_Standard.TON:=(PT:=T#1S);
	tonSys_InitTimeout			: Tc2_Standard.TON:=(PT:=T#20S);					
	tonFirstAutoCycle			: Tc2_Standard.TON:=(PT:=T#500MS);
	
/////////////////////////////////////////////////////////////////////////////////////PROCESS CYCLE/////////////////////////////////////////////////////////////////////////////////////	
	
	eCycleState					: E_ProcessCycle;
	tonCMD_Done					: TON;
	tonResetAllCMD				: TON;
	tonExecute					: TON;
	tonSave_Data				: TON;
	tonWriteToCsv				: TON;
	rNoAutoCycle				: R_TRIG;
	
	bStartProcessCondition		: BOOL;
	bIndexDataHistoryFlag		: BOOL;
	rIndexDataHistoryFlag		: R_TRIG;
	bPASS						: BOOL;
	bFAIL						: BOOL;
	i							: INT;
	

	
END_VAR

/////////////////////////////////////////////////////////////////////////////////////GENERAL/////////////////////////////////////////////////////////////////////////////////////
a_ACT_MachineStatus();
b_ACT_ProcessCycle();

ACTION a_ACT_MachineStatus:
/////////////////////////////////////////////////////////////////////////////////////TIMERS/////////////////////////////////////////////////////////////////////////////////////
tonSys_Init(IN:=stMachineStatus.bInitialising);
tonSys_InitTimeout(IN:=stMachineStatus.bInitialising);


/////////////////////////////////////////////////////////////////////////////////////CONDITIONS/////////////////////////////////////////////////////////////////////////////////////
				IF NOT stMasterCtrl.bNoImmediateFault THEN
					stMachineStatus.eMachineState 		:= E_MachineState.IMMEDIATE_FAULT;
				END_IF
				
				IF stMachineStatus.eMachineState		= E_MachineState.STOPPING OR
				stMachineStatus.eMachineState			= E_MachineState.IMMEDIATE_FAULT OR
				stMachineStatus.eMachineState			= E_MachineState.CYCLE_STOP_FAULT THEN
					
					CMD_Station1.bAbort					:= TRUE;	
					CMD_Station2.bAbort					:= TRUE;	
					CMD_Station3.bAbort					:= TRUE;
				
					CMD_Station1.bEnable				:= FALSE;
					CMD_Station2.bEnable				:= FALSE;
					CMD_Station3.bEnable				:= FALSE;
					
				END_IF
				
				IF 	stButtonsLamps.bResetButtonFallingEdge THEN
					CMD_Station1.bReset					:= TRUE;
					CMD_Station2.bReset					:= TRUE;
					CMD_Station3.bReset					:= TRUE;
				ELSE 
					CMD_Station1.bReset					:= FALSE;
					CMD_Station2.bReset					:= FALSE;
					CMD_Station3.bReset					:= FALSE;
				END_IF		
				
/////////////////////////////////////////////////////////////////////////////////////MACHINE CONTROL/////////////////////////////////////////////////////////////////////////////////////

CASE stMachineStatus.eMachineState OF

E_MachineState.SYSTEM_POWER_UP: 		

				IF tonSystemPowerUP.Q THEN
						stMachineStatus.eMachineState 	:= E_MachineState.IMMEDIATE_STOPPED;//
				END_IF
	
E_MachineState.IMMEDIATE_STOPPED:		

				IF stButtonsLamps.bResetButtonFallingEdge THEN
						stMachineStatus.eMachineState 	:= E_MachineState.SYSTEM_INITIALISING;//
				END_IF	


E_MachineState.SYSTEM_INITIALISING:		
				
				CMD_Station1.bAbort						:= FALSE;	
				CMD_Station2.bAbort						:= FALSE;	
				CMD_Station3.bAbort						:= FALSE;	

				IF tonSys_Init.Q THEN
					CMD_Station1.bEnable				:= TRUE;
					CMD_Station2.bEnable				:= TRUE;
					CMD_Station3.bEnable				:= TRUE;						
				END_IF

				IF B_1_1_PRG_Master_Station_1.STATUS.bReady AND B_2_1_PRG_Master_Station_2.STATUS.bReady AND B_3_1_PRG_Master_Station_3.STATUS.bReady THEN 
					stMachineStatus.eMachineState		:= E_MachineState.SYSTEM_READY_TO_START;
				ELSIF stButtonsLamps.bStopButtonFallingEdge OR  
				stMasterCtrl.bCycleStopRequest OR tonSys_InitTimeout.Q THEN
					stMachineStatus.eMachineState 		:= E_MachineState.STOPPING;	
				ELSIF NOT stMasterCtrl.bNoCycleStopFault THEN		
					stMachineStatus.eMachineState 		:= E_MachineState.CYCLE_STOP_FAULT;
				END_IF
			
					
E_MachineState.SYSTEM_READY_TO_START:	

				IF 	 stButtonsLamps.bStartButtonFallingEdge AND stMasterCtrl.bAllStationsReady THEN
					stMachineStatus.eMachineState 		:= E_MachineState.SYSTEM_AUTO_CYCLE;
				ELSIF stButtonsLamps.bStopButtonFallingEdge THEN
					stMachineStatus.eMachineState 		:= E_MachineState.STOPPING;		
				ELSIF stMasterCtrl.bNoCycleStopFault THEN	
					stMachineStatus.eMachineState 		:= E_MachineState.CYCLE_STOP_FAULT;
				ELSIF GVL_Master.stMasterCTRL.bManualModeRequest AND stMasterCtrl.bNoCycleStopFault THEN
					stMachineStatus.eMachineState 		:= E_MachineState.MANUAL_MODE;
				END_IF

				

E_MachineState.SYSTEM_AUTO_CYCLE:		

				IF stButtonsLamps.bStopButtonFallingEdge OR stMasterCtrl.bCycleStopRequest THEN					
					stMachineStatus.eMachineState 		:= E_MachineState.STOPPING;
				ELSIF NOT stMasterCtrl.bNoCycleStopFault THEN	
					stMachineStatus.eMachineState 		:= E_MachineState.CYCLE_STOP_FAULT;
				END_IF
				
E_MachineState.SYSTEM_STANDBY:



E_MachineState.STOPPING:	

				IF stMasterCtrl.bAllStationsStopped THEN
					stMachineStatus.eMachineState 		:= E_MachineState.CYCLE_STOPPED;
				ELSIF NOT stMasterCtrl.bNoCycleStopFault THEN	
					stMachineStatus.eMachineState 		:= E_MachineState.CYCLE_STOP_FAULT;					
				END_IF

E_MachineState.CYCLE_STOPPED:			

				IF stMasterCtrl.bNoCycleStopFault   AND NOT stMasterCtrl.bCycleStopRequest  AND stButtonsLamps.bResetButtonFallingEdge THEN	
					stMachineStatus.eMachineState 		:= E_MachineState.SYSTEM_INITIALISING;		
				END_IF	

E_MachineState.IMMEDIATE_FAULT:	
				
				IF stMasterCtrl.bNoImmediateFault	THEN
					stMachineStatus.eMachineState		:= E_MachineState.IMMEDIATE_STOPPED;		
				END_IF

E_MachineState.CYCLE_STOP_FAULT:		
				
				IF stMasterCtrl.bNoCycleStopFault AND stMasterCtrl.bAllStationsStopped THEN
					stMachineStatus.eMachineState 		:= E_MachineState.CYCLE_STOPPED;
				END_IF	


E_MachineState.MANUAL_MODE:

				IF stButtonsLamps.bStopButtonFallingEdge OR NOT GVL_Master.stMasterCTRL.bManualModeRequest THEN
					stMachineStatus.eMachineState 		:= E_MachineState.STOPPING;
				ELSIF  NOT stMasterCtrl.bNoCycleStopFault THEN	
					stMachineStatus.eMachineState 		:= E_MachineState.CYCLE_STOP_FAULT;								
				ELSE 
					CMD_Station1.bManualMode			:=TRUE;
					CMD_Station2.bManualMode			:=TRUE;
					CMD_Station3.bManualMode			:=TRUE;
				END_IF
ELSE
stMachineStatus.eMachineState:=E_MachineState.SYSTEM_POWER_UP;		
END_CASE									


/////////////////////////////////////////////////////////////////////////////////////MACHINE STATUS/////////////////////////////////////////////////////////////////////////////////////
stMachineStatus.bSystemPowerUp 			:= (stMachineStatus.eMachineState = E_MachineState.SYSTEM_POWER_UP);
stMachineStatus.bImmediateStopped 		:= (stMachineStatus.eMachineState = E_MachineState.IMMEDIATE_STOPPED);
stMachineStatus.bInitialising 			:= (stMachineStatus.eMachineState = E_MachineState.SYSTEM_INITIALISING);
stMachineStatus.bReadyToStart 			:= (stMachineStatus.eMachineState = E_MachineState.SYSTEM_READY_TO_START);
stMachineStatus.bAutoCycle 				:= (stMachineStatus.eMachineState = E_MachineState.SYSTEM_AUTO_CYCLE);
stMachineStatus.bStandby 				:= (stMachineStatus.eMachineState = E_MachineState.SYSTEM_STANDBY);
stMachineStatus.bStopping 				:= (stMachineStatus.eMachineState = E_MachineState.STOPPING);
stMachineStatus.bCycleStopped 			:= (stMachineStatus.eMachineState = E_MachineState.CYCLE_STOPPED);
stMachineStatus.bImmediateFault 		:= (stMachineStatus.eMachineState = E_MachineState.IMMEDIATE_FAULT);
stMachineStatus.bCycleStopFault 		:= (stMachineStatus.eMachineState = E_MachineState.CYCLE_STOP_FAULT);
stMachineStatus.bManualMode 			:= (stMachineStatus.eMachineState = E_MachineState.MANUAL_MODE);

/////////////////////////////////////////////////////////////////////////////////////FLAGS/////////////////////////////////////////////////////////////////////////////////////
stMasterCtrl.bAllStationsStopped		:= (B_1_1_PRG_Master_Station_1.STATUS.bReady AND B_2_1_PRG_Master_Station_2.STATUS.bReady AND B_3_1_PRG_Master_Station_3.STATUS.bReady ) OR
										   (NOT B_1_1_PRG_Master_Station_1.STATUS.bBusy AND NOT B_2_1_PRG_Master_Station_2.STATUS.bBusy AND NOT B_3_1_PRG_Master_Station_3.STATUS.bBusy );
										   
stMasterCtrl.bAllStationsReady			:= B_1_1_PRG_Master_Station_1.bReady AND B_2_1_PRG_Master_Station_2.bReady AND B_3_1_PRG_Master_Station_3.bReady;
END_ACTION

ACTION b_ACT_ProcessCycle:
/////////////////////////////////////////////////////////////////////////////////////UTILITIES & TRIGGERS/////////////////////////////////////////////////////////////////////////////////////

tonCMD_Done( IN := , PT := T#500MS);
tonSave_Data( IN :=  eCycleState = E_ProcessCycle.SAVE_DATA2, PT := T#500MS);
tonResetAllCMD( IN := eCycleState = E_ProcessCycle.RESET_ALL_CMD, PT := T#500MS);
tonWriteToCsv( IN := eCycleState = E_ProcessCycle.CSV, PT := T#500MS);

tonExecute( IN := 	eCycleState = E_ProcessCycle.STATION1_MOV1 OR
					eCycleState = E_ProcessCycle.STATION2_MOV2 OR
					eCycleState = E_ProcessCycle.STATION1_MOV3_STATION2_MOV2 OR
					eCycleState = E_ProcessCycle.STATION3_MOV3,
					PT := T#500MS);
				

rNoAutoCycle( CLK := stMachineStatus.bAutoCycle);

/////////////////////////////////////////////////////////////////////////////////////CONDITIONS/////////////////////////////////////////////////////////////////////////////////////

//bStartProcessCondition := ; //

IF rNoAutoCycle.Q THEN
	eCycleState												:= E_ProcessCycle.RESET_ALL_CMD;
END_IF


CASE eCycleState OF
	
E_ProcessCycle.RESET_ALL_CMD:

				stStation1.Mov1								:= FALSE;
				stStation1.Mov2								:= FALSE;
				stStation1.Mov3								:= FALSE;
				B_1_1_PRG_Master_Station_1.CMD.bExecute		:= FALSE;
				B_1_1_PRG_Master_Station_1.CMD.bReady 		:= FALSE;
				stStation2.Mov1								:= FALSE;
				stStation2.Mov2								:= FALSE;
				stStation2.Mov3								:= FALSE;
				B_2_1_PRG_Master_Station_2.CMD.bExecute		:= FALSE;
				B_2_1_PRG_Master_Station_2.CMD.bReady 		:= FALSE;
				stStation3.Mov1								:= FALSE;
				stStation3.Mov2								:= FALSE;
				stStation3.Mov3								:= FALSE;
				B_3_1_PRG_Master_Station_3.CMD.bExecute		:= FALSE;
				B_3_1_PRG_Master_Station_3.CMD.bReady 		:= FALSE;
				stCSVProcess.bWriteData						:= FALSE;
				
				//bIndexDataHistoryFlag						:= FALSE;
				
				
				IF tonResetAllCMD.Q AND stMachineStatus.bAutoCycle THEN
					eCycleState								:= E_ProcessCycle.IDLE;						
				END_IF
	
E_ProcessCycle.IDLE:
				
				IF bStartProcessCondition AND B_1_1_PRG_Master_Station_1.STATUS.bReady THEN
					eCycleState								:= E_ProcessCycle.STATION1_MOV1;
				END_IF
							
E_ProcessCycle.STATION1_MOV1:

				stStation1.Mov1								:= TRUE;
				B_1_1_PRG_Master_Station_1.CMD.bExecute		:= TRUE;
				
